C07312=1184.662,313.073,-71.587,-176.592,7.819,148.515
C07313=1184.666,312.825,-71.556,-176.595,7.816,148.515
C07314=1184.670,312.577,-71.525,-176.597,7.813,148.515
C07315=1184.675,312.329,-71.495,-176.599,7.810,148.515
C07316=1184.679,312.081,-71.463,-176.602,7.807,148.515
C07317=1184.683,311.833,-71.432,-176.604,7.804,148.515
C07318=1184.687,311.585,-71.402,-176.607,7.801,148.514
C07319=1184.692,311.337,-71.371,-176.609,7.798,148.515
C07320=1184.696,311.089,-71.340,-176.612,7.795,148.515
C07321=1184.700,310.841,-71.309,-176.615,7.792,148.515
C07322=1184.704,310.593,-71.279,-176.617,7.790,148.514
C07323=1184.709,310.345,-71.248,-176.619,7.787,148.514
C07324=1184.713,310.096,-71.217,-176.622,7.784,148.514
C07325=1184.717,309.849,-71.187,-176.624,7.780,148.514
C07326=1184.721,309.601,-71.156,-176.627,7.777,148.514
C07327=1184.726,309.353,-71.125,-176.630,7.774,148.514
C07328=1184.729,309.104,-71.095,-176.632,7.771,148.514
C07329=1184.734,308.856,-71.064,-176.634,7.769,148.514
C07330=1184.739,308.608,-71.034,-176.637,7.766,148.514
C07331=1184.742,308.360,-71.004,-176.640,7.763,148.514
C07332=1184.746,308.112,-70.973,-176.642,7.760,148.514
C07333=1184.751,307.864,-70.942,-176.645,7.757,148.514
C07334=1184.755,307.616,-70.912,-176.647,7.754,148.514
C07335=1184.760,307.368,-70.881,-176.650,7.751,148.514
C07336=1184.764,307.119,-70.850,-176.652,7.748,148.514
C07337=1184.768,306.871,-70.820,-176.654,7.745,148.514
C07338=1184.772,306.623,-70.790,-176.657,7.742,148.514
C07339=1184.776,306.375,-70.760,-176.660,7.739,148.514
C07340=1184.781,306.128,-70.729,-176.662,7.736,148.514
C07341=1184.785,305.879,-70.698,-176.665,7.733,148.514
C07342=1184.789,305.631,-70.668,-176.667,7.731,148.514
C07343=1184.794,305.383,-70.637,-176.670,7.728,148.514
C07344=1184.798,305.135,-70.607,-176.672,7.725,148.514
C07345=1184.802,304.886,-70.577,-176.675,7.722,148.514
C07346=1184.806,304.638,-70.547,-176.677,7.718,148.514
C07347=1184.810,304.390,-70.516,-176.680,7.715,148.514
C07348=1184.814,304.142,-70.486,-176.682,7.713,148.514
C07349=1184.819,303.894,-70.456,-176.685,7.710,148.514
C07350=1184.823,303.646,-70.426,-176.688,7.707,148.514
C07351=1184.828,303.398,-70.395,-176.690,7.704,148.514
C07352=1184.832,303.150,-70.365,-176.693,7.701,148.514
C07353=1184.836,302.901,-70.334,-176.695,7.698,148.514
C07354=1184.840,302.653,-70.305,-176.697,7.696,148.514
C07355=1184.845,302.405,-70.274,-176.700,7.693,148.514
C07356=1184.849,302.157,-70.244,-176.702,7.689,148.514
C07357=1184.853,301.909,-70.214,-176.705,7.686,148.514
C07358=1184.857,301.661,-70.184,-176.708,7.683,148.514
C07359=1184.861,301.413,-70.154,-176.711,7.680,148.514
C07360=1184.866,301.165,-70.123,-176.713,7.678,148.514
C07361=1184.870,300.916,-70.094,-176.715,7.675,148.514
C07362=1184.874,300.668,-70.063,-176.718,7.672,148.513
C07363=1184.878,300.420,-70.033,-176.720,7.669,148.513
C07364=1184.882,300.172,-70.003,-176.723,7.666,148.513
C07365=1184.887,299.924,-69.973,-176.725,7.664,148.514
C07366=1184.891,299.675,-69.944,-176.728,7.661,148.514
C07367=1184.895,299.428,-69.913,-176.731,7.658,148.514
C07368=1184.900,299.179,-69.883,-176.733,7.655,148.514
C07369=1184.904,298.931,-69.853,-176.736,7.651,148.513
C07370=1184.908,298.683,-69.824,-176.738,7.648,148.513
C07371=1184.913,298.435,-69.794,-176.741,7.646,148.514
C07372=1184.917,298.187,-69.764,-176.743,7.643,148.514
C07373=1184.921,297.939,-69.734,-176.746,7.640,148.514
C07374=1184.926,297.690,-69.704,-176.749,7.637,148.514
C07375=1184.930,297.442,-69.674,-176.751,7.634,148.514
C07376=1184.934,297.194,-69.644,-176.753,7.632,148.513
C07377=1184.938,296.946,-69.615,-176.756,7.629,148.514
C07378=1184.943,296.698,-69.584,-176.759,7.626,148.514
C07379=1184.947,296.450,-69.555,-176.761,7.623,148.514
C07380=1184.951,296.201,-69.525,-176.763,7.621,148.514
C07381=1184.956,295.953,-69.496,-176.766,7.618,148.514
C07382=1184.960,295.705,-69.465,-176.769,7.615,148.514
C07383=1184.964,295.457,-69.436,-176.772,7.612,148.514
C07384=1184.969,295.209,-69.406,-176.774,7.609,148.514
C07385=1184.973,294.960,-69.377,-176.776,7.606,148.514
C07386=1184.977,294.713,-69.347,-176.779,7.603,148.514
C07387=1184.981,294.464,-69.317,-176.781,7.600,148.514
C07388=1184.986,294.216,-69.287,-176.784,7.597,148.514
C07389=1184.990,293.968,-69.258,-176.787,7.594,148.514
C07390=1184.994,293.719,-69.228,-176.789,7.592,148.514
C07391=1184.998,293.471,-69.199,-176.792,7.589,148.514
C07392=1185.002,293.223,-69.169,-176.794,7.586,148.514
C07393=1185.007,292.975,-69.140,-176.797,7.583,148.514
C07394=1185.011,292.727,-69.109,-176.799,7.581,148.514
C07395=1185.015,292.478,-69.080,-176.802,7.578,148.514
C07396=1185.020,292.230,-69.050,-176.805,7.575,148.514
C07397=1185.024,291.982,-69.021,-176.807,7.571,148.514
C07398=1185.028,291.734,-68.991,-176.810,7.568,148.514
C07399=1185.032,291.485,-68.962,-176.812,7.566,148.514
C07400=1185.036,291.237,-68.932,-176.815,7.563,148.514
C07401=1185.040,290.989,-68.903,-176.817,7.560,148.514
C07402=1185.045,290.741,-68.874,-176.820,7.557,148.514
C07403=1185.049,290.493,-68.844,-176.822,7.555,148.514
C07404=1185.054,290.245,-68.815,-176.825,7.552,148.514
C07405=1185.058,289.996,-68.785,-176.828,7.549,148.514
C07406=1185.062,289.748,-68.756,-176.830,7.546,148.514
C07407=1185.066,289.499,-68.727,-176.833,7.544,148.514
C07408=1185.071,289.251,-68.698,-176.835,7.541,148.514
C07409=1185.075,289.003,-68.668,-176.838,7.538,148.514
C07410=1185.080,288.729,-68.635,-176.841,7.535,148.514
C07411=1185.084,288.454,-68.603,-176.843,7.532,148.514
C07412=1185.090,288.179,-68.571,-176.846,7.529,148.514
C07413=1185.094,287.905,-68.539,-176.849,7.525,148.514
C07414=1185.098,287.657,-68.509,-176.852,7.523,148.514
C07415=1185.103,287.408,-68.481,-176.854,7.520,148.514
C07416=1185.107,287.160,-68.451,-176.857,7.517,148.514
C07417=1185.111,286.911,-68.422,-176.860,7.514,148.514
C07418=1185.116,286.663,-68.392,-176.862,7.512,148.515
C07419=1185.120,286.416,-68.363,-176.865,7.509,148.515
C07420=1185.125,286.167,-68.334,-176.867,7.506,148.515
C07421=1185.129,285.918,-68.305,-176.869,7.504,148.515
C07422=1185.133,285.670,-68.275,-176.872,7.501,148.515
C07423=1185.138,285.421,-68.247,-176.875,7.498,148.515
C07424=1185.142,285.174,-68.218,-176.878,7.495,148.515
C07425=1185.146,284.926,-68.189,-176.880,7.493,148.515
C07426=1185.150,284.677,-68.160,-176.883,7.490,148.515
C07427=1185.155,284.429,-68.131,-176.885,7.487,148.515
C07428=1185.159,284.181,-68.102,-176.888,7.484,148.515
C07429=1185.164,283.932,-68.073,-176.890,7.481,148.515
C07430=1185.167,283.684,-68.044,-176.893,7.478,148.515
C07431=1185.171,283.436,-68.014,-176.896,7.475,148.515
C07432=1185.177,283.188,-67.986,-176.898,7.472,148.515
C07433=1185.181,282.940,-67.957,-176.900,7.470,148.515
C07434=1185.185,282.691,-67.928,-176.903,7.467,148.515
C07435=1185.189,282.442,-67.898,-176.906,7.464,148.515
C07436=1185.194,282.195,-67.871,-176.908,7.462,148.515
C07437=1185.198,281.946,-67.841,-176.911,7.459,148.515
C07438=1185.202,281.697,-67.812,-176.914,7.456,148.515
C07439=1185.207,281.450,-67.783,-176.916,7.453,148.515
C07440=1185.211,281.201,-67.755,-176.918,7.451,148.516
C07441=1185.215,280.953,-67.726,-176.921,7.448,148.516
C07442=1185.220,280.705,-67.697,-176.924,7.445,148.516
C07443=1185.224,280.457,-67.669,-176.926,7.443,148.516
C07444=1185.228,280.208,-67.640,-176.929,7.440,148.516
C07445=1185.232,279.960,-67.610,-176.932,7.437,148.516
C07446=1185.237,279.711,-67.582,-176.934,7.435,148.516
C07447=1185.241,279.463,-67.554,-176.937,7.432,148.516
C07448=1185.245,279.215,-67.524,-176.940,7.429,148.516
C07449=1185.250,278.966,-67.496,-176.942,7.426,148.516
C07450=1185.254,278.718,-67.467,-176.944,7.424,148.516
C07451=1185.258,278.470,-67.438,-176.947,7.421,148.516
C07452=1185.263,278.222,-67.411,-176.950,7.418,148.516
C07453=1185.267,277.973,-67.381,-176.952,7.416,148.516
C07454=1185.272,277.725,-67.353,-176.955,7.413,148.516
C07455=1185.276,277.477,-67.325,-176.957,7.410,148.516
C07456=1185.280,277.228,-67.296,-176.960,7.408,148.517
C07457=1185.285,276.980,-67.267,-176.962,7.405,148.517
C07458=1185.289,276.732,-67.239,-176.965,7.402,148.517
C07459=1185.293,276.483,-67.210,-176.968,7.400,148.517
C07460=1185.298,276.235,-67.182,-176.970,7.397,148.517
C07461=1185.302,275.987,-67.153,-176.973,7.394,148.517
C07462=1185.306,275.739,-67.125,-176.975,7.392,148.517
C07463=1185.311,275.490,-67.096,-176.978,7.389,148.517
C07464=1185.314,275.241,-67.068,-176.981,7.386,148.517
C07465=1185.319,274.993,-67.040,-176.983,7.384,148.517
C07466=1185.324,274.745,-67.010,-176.986,7.381,148.517
C07467=1185.328,274.497,-66.983,-176.988,7.378,148.517
C07468=1185.332,274.248,-66.954,-176.991,7.375,148.517
C07469=1185.337,274.000,-66.926,-176.994,7.373,148.518
C07470=1185.341,273.751,-66.897,-176.996,7.370,148.518
C07471=1185.345,273.503,-66.869,-176.999,7.368,148.518
C07472=1185.350,273.255,-66.841,-177.001,7.365,148.518
C07473=1185.354,273.006,-66.813,-177.004,7.362,148.518
C07474=1185.358,272.758,-66.785,-177.006,7.359,148.518
C07475=1185.363,272.509,-66.756,-177.009,7.356,148.518
C07476=1185.367,272.261,-66.728,-177.012,7.353,148.518
C07477=1185.371,272.013,-66.699,-177.014,7.351,148.518
C07478=1185.376,271.765,-66.671,-177.017,7.349,148.518
C07479=1185.380,271.516,-66.642,-177.020,7.346,148.518
C07480=1185.385,271.268,-66.615,-177.022,7.343,148.519
C07481=1185.389,271.019,-66.587,-177.025,7.340,148.519
C07482=1185.394,270.771,-66.559,-177.027,7.337,148.519
C07483=1185.397,270.522,-66.531,-177.029,7.335,148.519
C07484=1185.402,270.274,-66.502,-177.032,7.332,148.519
C07485=1185.406,270.026,-66.474,-177.035,7.330,148.519
C07486=1185.411,269.778,-66.446,-177.038,7.328,148.519
C07487=1185.415,269.529,-66.418,-177.040,7.325,148.519
C07488=1185.419,269.281,-66.390,-177.042,7.322,148.519
C07489=1185.423,269.032,-66.362,-177.045,7.319,148.519
C07490=1185.428,268.784,-66.333,-177.048,7.316,148.519
C07491=1185.433,268.536,-66.306,-177.051,7.315,148.520
C07492=1185.437,268.287,-66.278,-177.053,7.312,148.520
C07493=1185.442,268.039,-66.250,-177.056,7.309,148.520
C07494=1185.445,267.790,-66.222,-177.058,7.306,148.520
C07495=1185.450,267.543,-66.194,-177.061,7.303,148.520
C07496=1185.455,267.293,-66.166,-177.063,7.301,148.520
C07497=1185.459,267.045,-66.138,-177.066,7.299,148.520
C07498=1185.463,266.797,-66.110,-177.069,7.296,148.520
C07499=1185.467,266.549,-66.082,-177.071,7.293,148.520
C07500=1185.472,266.300,-66.054,-177.074,7.290,148.520
C07501=1185.476,266.051,-66.026,-177.077,7.287,148.520
C07502=1185.481,265.803,-65.999,-177.079,7.285,148.520
C07503=1185.485,265.556,-65.971,-177.082,7.283,148.521
C07504=1185.490,265.306,-65.943,-177.084,7.281,148.521
C07505=1185.494,265.058,-65.915,-177.087,7.278,148.521
C07506=1185.498,264.810,-65.887,-177.090,7.275,148.521
C07507=1185.502,264.561,-65.860,-177.092,7.272,148.521
C07508=1185.507,264.313,-65.832,-177.095,7.270,148.521
C07509=1185.512,264.064,-65.804,-177.097,7.268,148.521
C07510=1185.516,263.816,-65.776,-177.100,7.265,148.521
C07511=1185.520,263.568,-65.748,-177.103,7.262,148.521
C07512=1185.524,263.319,-65.721,-177.105,7.259,148.522
C07513=1185.529,263.071,-65.693,-177.108,7.257,148.522
C07514=1185.534,262.798,-65.663,-177.111,7.254,148.522
C07515=1185.539,262.525,-65.632,-177.113,7.251,148.522
C07516=1185.544,262.252,-65.602,-177.117,7.248,148.522
C07517=1185.548,261.979,-65.572,-177.119,7.245,148.522
C07518=1185.552,261.731,-65.545,-177.121,7.243,148.522
C07519=1185.557,261.482,-65.516,-177.125,7.240,148.523
C07520=1185.562,261.233,-65.489,-177.127,7.238,148.523
C07521=1185.566,260.986,-65.461,-177.130,7.235,148.523
C07522=1185.571,260.737,-65.434,-177.132,7.233,148.523
C07523=1185.574,260.489,-65.406,-177.134,7.230,148.523
C07524=1185.579,260.240,-65.379,-177.138,7.227,148.523
C07525=1185.584,259.992,-65.352,-177.140,7.225,148.523
C07526=1185.587,259.743,-65.324,-177.143,7.222,148.523
C07527=1185.592,259.494,-65.297,-177.145,7.220,148.523
C07528=1185.596,259.247,-65.269,-177.148,7.217,148.524
C07529=1185.601,258.998,-65.242,-177.150,7.215,148.524
C07530=1185.605,258.749,-65.214,-177.153,7.212,148.524
C07531=1185.610,258.501,-65.187,-177.156,7.210,148.524
C07532=1185.614,258.253,-65.160,-177.158,7.207,148.524
C07533=1185.619,258.004,-65.132,-177.161,7.204,148.524
C07534=1185.623,257.755,-65.104,-177.163,7.202,148.524
C07535=1185.627,257.507,-65.077,-177.166,7.200,148.525
C07536=1185.632,257.258,-65.050,-177.168,7.198,148.525
C07537=1185.637,257.010,-65.023,-177.171,7.195,148.525
C07538=1185.641,256.762,-64.995,-177.173,7.192,148.525
C07539=1185.645,256.513,-64.968,-177.176,7.190,148.525
C07540=1185.650,256.264,-64.941,-177.179,7.187,148.525
C07541=1185.654,256.016,-64.914,-177.181,7.185,148.525
C07542=1185.658,255.768,-64.887,-177.185,7.182,148.525
C07543=1185.663,255.520,-64.860,-177.187,7.180,148.526
C07544=1185.667,255.271,-64.832,-177.189,7.177,148.526
C07545=1185.671,255.022,-64.805,-177.192,7.175,148.526
C07546=1185.676,254.774,-64.778,-177.195,7.172,148.526
C07547=1185.681,254.525,-64.751,-177.197,7.170,148.526
C07548=1185.685,254.277,-64.724,-177.200,7.167,148.526
C07549=1185.689,254.028,-64.696,-177.202,7.165,148.526
C07550=1185.693,253.780,-64.669,-177.205,7.162,148.526
C07551=1185.698,253.531,-64.642,-177.207,7.160,148.527
C07552=1185.702,253.283,-64.615,-177.210,7.157,148.527
C07553=1185.707,253.034,-64.588,-177.213,7.155,148.527
C07554=1185.712,252.786,-64.561,-177.215,7.152,148.527
C07555=1185.715,252.538,-64.535,-177.218,7.150,148.527
C07556=1185.719,252.289,-64.507,-177.221,7.147,148.527
C07557=1185.724,252.040,-64.480,-177.223,7.145,148.527
C07558=1185.729,251.792,-64.453,-177.226,7.142,148.528
C07559=1185.733,251.543,-64.426,-177.229,7.139,148.528
C07560=1185.737,251.295,-64.399,-177.231,7.137,148.528
C07561=1185.742,251.046,-64.372,-177.234,7.135,148.528
C07562=1185.747,250.798,-64.345,-177.236,7.132,148.528
C07563=1185.751,250.549,-64.318,-177.239,7.130,148.528
C07564=1185.755,250.301,-64.292,-177.242,7.128,148.529
C07565=1185.760,250.053,-64.265,-177.244,7.125,148.529
C07566=1185.765,249.804,-64.238,-177.247,7.123,148.529
C07567=1185.768,249.555,-64.211,-177.250,7.120,148.529
C07568=1185.773,249.306,-64.185,-177.252,7.118,148.529
C07569=1185.778,249.058,-64.157,-177.255,7.115,148.529
C07570=1185.781,248.810,-64.131,-177.257,7.113,148.530
C07571=1185.786,248.561,-64.104,-177.260,7.111,148.530
C07572=1185.791,248.313,-64.077,-177.262,7.108,148.530
C07573=1185.795,248.064,-64.050,-177.265,7.106,148.530
C07574=1185.799,247.816,-64.023,-177.268,7.103,148.530
C07575=1185.804,247.567,-63.997,-177.270,7.101,148.530
C07576=1185.808,247.319,-63.971,-177.273,7.098,148.530
C07577=1185.813,247.070,-63.943,-177.275,7.096,148.531
C07578=1185.818,246.822,-63.916,-177.278,7.093,148.531
C07579=1185.822,246.573,-63.891,-177.281,7.091,148.531
C07580=1185.826,246.324,-63.864,-177.283,7.088,148.531
C07581=1185.830,246.076,-63.837,-177.286,7.086,148.531
C07582=1185.835,245.828,-63.810,-177.289,7.083,148.531
C07583=1185.840,245.578,-63.784,-177.291,7.082,148.532
C07584=1185.844,245.330,-63.757,-177.294,7.079,148.532
C07585=1185.849,245.082,-63.730,-177.296,7.076,148.532
C07586=1185.853,244.833,-63.704,-177.299,7.074,148.532
C07587=1185.857,244.584,-63.677,-177.302,7.072,148.532
C07588=1185.861,244.336,-63.651,-177.305,7.069,148.533
C07589=1185.866,244.087,-63.625,-177.307,7.067,148.533
C07590=1185.870,243.839,-63.598,-177.309,7.065,148.533
C07591=1185.875,243.590,-63.572,-177.312,7.062,148.533
C07592=1185.879,243.342,-63.545,-177.315,7.060,148.533
C07593=1185.884,243.093,-63.518,-177.318,7.057,148.533
C07594=1185.888,242.844,-63.492,-177.320,7.055,148.533
C07595=1185.893,242.596,-63.465,-177.323,7.052,148.534
C07596=1185.897,242.348,-63.440,-177.325,7.050,148.534
C07597=1185.902,242.099,-63.413,-177.328,7.047,148.534
C07598=1185.906,241.850,-63.387,-177.331,7.045,148.534
C07599=1185.911,241.602,-63.360,-177.333,7.043,148.534
C07600=1185.915,241.353,-63.334,-177.336,7.041,148.535
C07601=1185.920,241.105,-63.307,-177.338,7.039,148.535
C07602=1185.924,240.856,-63.282,-177.341,7.036,148.535
C07603=1185.928,240.608,-63.255,-177.344,7.034,148.535
C07604=1185.933,240.359,-63.229,-177.346,7.031,148.535
C07605=1185.937,240.110,-63.202,-177.349,7.029,148.535
C07606=1185.942,239.862,-63.176,-177.352,7.026,148.536
C07607=1185.947,239.613,-63.151,-177.354,7.024,148.536
C07608=1185.951,239.365,-63.124,-177.357,7.022,148.536
C07609=1185.956,239.116,-63.098,-177.360,7.019,148.536
C07610=1185.959,238.868,-63.071,-177.362,7.017,148.536
C07611=1185.964,238.619,-63.046,-177.365,7.015,148.537
C07612=1185.969,238.370,-63.019,-177.367,7.012,148.537
C07613=1185.973,238.122,-62.993,-177.370,7.011,148.537
C07614=1185.977,237.874,-62.967,-177.373,7.008,148.537
C07615=1185.982,237.624,-62.941,-177.375,7.005,148.537
C07616=1185.986,237.376,-62.915,-177.378,7.003,148.538
C07617=1185.991,237.127,-62.889,-177.380,7.001,148.538
C07618=1185.996,236.855,-62.860,-177.383,6.998,148.538
C07619=1186.001,236.585,-62.832,-177.387,6.995,148.538
C07620=1186.006,236.313,-62.804,-177.389,6.993,148.538
C07621=1186.010,236.041,-62.775,-177.392,6.991,148.539
C07622=1186.015,235.792,-62.749,-177.394,6.988,148.539
C07623=1186.019,235.543,-62.723,-177.397,6.986,148.539
C07624=1186.024,235.295,-62.698,-177.400,6.984,148.539
C07625=1186.028,235.047,-62.671,-177.403,6.981,148.539
C07626=1186.033,234.798,-62.645,-177.405,6.979,148.539
C07627=1186.037,234.549,-62.619,-177.408,6.977,148.540
C07628=1186.042,234.301,-62.594,-177.410,6.974,148.540
C07629=1186.046,234.052,-62.568,-177.413,6.972,148.540
C07630=1186.050,233.804,-62.542,-177.415,6.970,148.540
C07631=1186.055,233.554,-62.516,-177.418,6.967,148.541
C07632=1186.060,233.307,-62.490,-177.421,6.965,148.541
C07633=1186.064,233.058,-62.464,-177.424,6.963,148.541
C07634=1186.068,232.809,-62.438,-177.426,6.961,148.541
C07635=1186.073,232.561,-62.412,-177.429,6.959,148.541
C07636=1186.077,232.312,-62.387,-177.432,6.956,148.542
C07637=1186.082,232.063,-62.361,-177.434,6.954,148.542
C07638=1186.087,231.815,-62.335,-177.437,6.952,148.542
C07639=1186.091,231.566,-62.309,-177.439,6.949,148.542
C07640=1186.096,231.318,-62.284,-177.442,6.947,148.543
C07641=1186.100,231.069,-62.258,-177.445,6.944,148.543
C07642=1186.104,230.820,-62.232,-177.447,6.942,148.543
C07643=1186.109,230.572,-62.207,-177.450,6.940,148.543
C07644=1186.113,230.323,-62.181,-177.453,6.938,148.543
C07645=1186.118,230.074,-62.155,-177.455,6.936,148.543
C07646=1186.123,229.826,-62.129,-177.458,6.934,148.544
C07647=1186.127,229.577,-62.104,-177.461,6.931,148.544
C07648=1186.131,229.328,-62.078,-177.463,6.929,148.544
C07649=1186.136,229.080,-62.052,-177.466,6.927,148.544
C07650=1186.141,228.831,-62.027,-177.468,6.924,148.545
C07651=1186.145,228.582,-62.002,-177.471,6.922,148.545
C07652=1186.150,228.334,-61.976,-177.474,6.919,148.545
C07653=1186.154,228.085,-61.951,-177.476,6.918,148.545
C07654=1186.158,227.836,-61.925,-177.479,6.916,148.546
C07655=1186.163,227.588,-61.899,-177.482,6.913,148.546
C07656=1186.167,227.339,-61.874,-177.484,6.911,148.546
C07657=1186.172,227.090,-61.849,-177.487,6.909,148.546
C07658=1186.177,226.842,-61.823,-177.490,6.906,148.546
C07659=1186.181,226.593,-61.798,-177.492,6.904,148.547
C07660=1186.186,226.345,-61.772,-177.495,6.902,148.547
C07661=1186.190,226.095,-61.747,-177.498,6.900,148.547
C07662=1186.194,225.847,-61.721,-177.500,6.897,148.547
C07663=1186.199,225.599,-61.696,-177.503,6.896,148.548
C07664=1186.203,225.350,-61.670,-177.505,6.893,148.548
C07665=1186.208,225.101,-61.646,-177.508,6.891,148.548
C07666=1186.212,224.853,-61.620,-177.511,6.889,148.548
C07667=1186.216,224.604,-61.595,-177.513,6.886,148.548
C07668=1186.221,224.355,-61.570,-177.516,6.884,148.549
C07669=1186.226,224.106,-61.544,-177.518,6.882,148.549
C07670=1186.230,223.858,-61.519,-177.521,6.879,148.549
C07671=1186.235,223.609,-61.494,-177.524,6.878,148.549
C07672=1186.240,223.361,-61.468,-177.526,6.875,148.550
C07673=1186.244,223.112,-61.443,-177.529,6.874,148.550
C07674=1186.248,222.863,-61.418,-177.532,6.871,148.550
C07675=1186.253,222.615,-61.393,-177.534,6.869,148.550
C07676=1186.257,222.365,-61.368,-177.537,6.867,148.551
C07677=1186.262,222.117,-61.342,-177.540,6.864,148.551
C07678=1186.266,221.868,-61.317,-177.542,6.862,148.551
C07679=1186.271,221.620,-61.292,-177.545,6.860,148.551
C07680=1186.275,221.371,-61.267,-177.548,6.857,148.551
C07681=1186.280,221.122,-61.242,-177.550,6.856,148.552
C07682=1186.284,220.873,-61.216,-177.553,6.854,148.552
C07683=1186.289,220.625,-61.192,-177.556,6.851,148.552
C07684=1186.293,220.376,-61.167,-177.558,6.849,148.553
C07685=1186.298,220.128,-61.142,-177.561,6.847,148.553
C07686=1186.302,219.879,-61.116,-177.563,6.845,148.553
C07687=1186.307,219.630,-61.091,-177.567,6.842,148.553
C07688=1186.311,219.381,-61.067,-177.569,6.840,148.553
C07689=1186.316,219.133,-61.042,-177.571,6.838,148.554
C07690=1186.321,218.883,-61.017,-177.575,6.836,148.554
C07691=1186.325,218.635,-60.991,-177.577,6.834,148.554
C07692=1186.329,218.386,-60.967,-177.579,6.832,148.555
C07693=1186.334,218.138,-60.941,-177.582,6.830,148.555
C07694=1186.338,217.889,-60.916,-177.585,6.827,148.555
C07695=1186.343,217.640,-60.892,-177.587,6.825,148.555
C07696=1186.348,217.392,-60.867,-177.590,6.824,148.556
C07697=1186.352,217.143,-60.842,-177.593,6.821,148.556
C07698=1186.357,216.894,-60.818,-177.596,6.819,148.556
C07699=1186.361,216.645,-60.792,-177.598,6.817,148.556
C07700=1186.366,216.397,-60.767,-177.600,6.815,148.556
C07701=1186.370,216.148,-60.743,-177.604,6.812,148.557
C07702=1186.375,215.899,-60.718,-177.606,6.810,148.557
C07703=1186.380,215.651,-60.693,-177.609,6.809,148.557
C07704=1186.384,215.402,-60.668,-177.611,6.806,148.558
C07705=1186.389,215.153,-60.644,-177.614,6.804,148.558
C07706=1186.392,214.904,-60.619,-177.617,6.802,148.558
C07707=1186.397,214.656,-60.594,-177.619,6.800,148.558
C07708=1186.402,214.407,-60.569,-177.622,6.797,148.559
C07709=1186.406,214.158,-60.545,-177.625,6.795,148.559
C07710=1186.411,213.909,-60.520,-177.627,6.793,148.559
C07711=1186.416,213.661,-60.496,-177.630,6.791,148.559
C07712=1186.420,213.412,-60.470,-177.633,6.789,148.560
C07713=1186.424,213.164,-60.446,-177.636,6.787,148.560
C07714=1186.429,212.914,-60.421,-177.638,6.785,148.560
C07715=1186.434,212.665,-60.397,-177.641,6.783,148.561
C07716=1186.438,212.417,-60.373,-177.644,6.780,148.561
C07717=1186.443,212.168,-60.347,-177.646,6.778,148.561
C07718=1186.447,211.919,-60.323,-177.649,6.776,148.561
C07719=1186.452,211.670,-60.299,-177.651,6.775,148.562
C07720=1186.456,211.421,-60.274,-177.654,6.772,148.562
C07721=1186.461,211.173,-60.250,-177.657,6.770,148.562
C07722=1186.466,210.903,-60.223,-177.659,6.768,148.562
C07723=1186.471,210.633,-60.197,-177.663,6.765,148.563
C07724=1186.476,210.362,-60.170,-177.665,6.764,148.563
C07725=1186.481,210.092,-60.143,-177.668,6.761,148.563
C07726=1186.485,209.843,-60.119,-177.671,6.759,148.563
C07727=1186.490,209.594,-60.094,-177.673,6.757,148.564
C07728=1186.494,209.345,-60.070,-177.676,6.754,148.564
C07729=1186.499,209.097,-60.045,-177.679,6.753,148.564
C07730=1186.504,208.848,-60.021,-177.681,6.750,148.565
C07731=1186.508,208.599,-59.996,-177.684,6.749,148.565
C07732=1186.513,208.350,-59.973,-177.687,6.747,148.565
C07733=1186.517,208.101,-59.949,-177.690,6.744,148.566
C07734=1186.522,207.853,-59.924,-177.692,6.742,148.566
C07735=1186.526,207.603,-59.899,-177.695,6.740,148.566
C07736=1186.531,207.355,-59.875,-177.697,6.738,148.566
C07737=1186.536,207.106,-59.851,-177.700,6.737,148.567
C07738=1186.540,206.858,-59.827,-177.703,6.734,148.567
C07739=1186.545,206.608,-59.802,-177.705,6.732,148.567
C07740=1186.549,206.359,-59.778,-177.708,6.730,148.567
C07741=1186.554,206.111,-59.754,-177.711,6.728,148.568
C07742=1186.559,205.862,-59.730,-177.713,6.725,148.568
C07743=1186.563,205.614,-59.705,-177.716,6.724,148.568
C07744=1186.567,205.365,-59.681,-177.719,6.722,148.569
C07745=1186.572,205.115,-59.657,-177.721,6.720,148.569
C07746=1186.577,204.867,-59.633,-177.724,6.718,148.569
C07747=1186.581,204.619,-59.609,-177.727,6.715,148.569
C07748=1186.586,204.370,-59.585,-177.730,6.713,148.570
C07749=1186.590,204.120,-59.561,-177.732,6.712,148.570
C07750=1186.595,203.872,-59.536,-177.735,6.710,148.570
C07751=1186.599,203.623,-59.512,-177.737,6.708,148.571
C07752=1186.604,203.374,-59.489,-177.740,6.706,148.571
C07753=1186.609,203.126,-59.464,-177.743,6.703,148.571
C07754=1186.613,202.876,-59.440,-177.746,6.701,148.572
C07755=1186.617,202.627,-59.417,-177.748,6.699,148.572
C07756=1186.622,202.379,-59.392,-177.750,6.697,148.572
C07757=1186.626,202.131,-59.368,-177.753,6.696,148.572
C07758=1186.632,201.881,-59.344,-177.756,6.693,148.573
C07759=1186.636,201.633,-59.320,-177.759,6.691,148.573
C07760=1186.641,201.384,-59.296,-177.761,6.689,148.573
C07761=1186.645,201.135,-59.273,-177.764,6.687,148.573
C07762=1186.649,200.886,-59.248,-177.766,6.685,148.574
C07763=1186.654,200.637,-59.225,-177.769,6.684,148.574
C07764=1186.659,200.389,-59.200,-177.772,6.681,148.574
C07765=1186.664,200.139,-59.177,-177.775,6.679,148.575
C07766=1186.668,199.891,-59.153,-177.777,6.677,148.575
C07767=1186.673,199.642,-59.130,-177.780,6.675,148.575
C07768=1186.677,199.394,-59.106,-177.783,6.674,148.576
C07769=1186.682,199.145,-59.082,-177.785,6.672,148.576
C07770=1186.686,198.896,-59.058,-177.788,6.669,148.576
C07771=1186.690,198.646,-59.034,-177.791,6.667,148.576
C07772=1186.695,198.398,-59.010,-177.793,6.665,148.577
C07773=1186.700,198.149,-58.986,-177.796,6.663,148.577
C07774=1186.704,197.900,-58.962,-177.799,6.662,148.577
C07775=1186.709,197.651,-58.939,-177.801,6.659,148.578
C07776=1186.714,197.403,-58.915,-177.803,6.658,148.578
C07777=1186.718,197.154,-58.892,-177.807,6.655,148.578
C07778=1186.723,196.905,-58.868,-177.809,6.653,148.579
C07779=1186.727,196.656,-58.844,-177.812,6.651,148.579
C07780=1186.732,196.407,-58.821,-177.815,6.650,148.579
C07781=1186.737,196.158,-58.797,-177.817,6.647,148.579
C07782=1186.741,195.910,-58.773,-177.820,6.646,148.580
C07783=1186.746,195.661,-58.750,-177.822,6.644,148.580
C07784=1186.751,195.412,-58.727,-177.825,6.642,148.580
C07785=1186.755,195.163,-58.703,-177.828,6.639,148.581
C07786=1186.760,194.914,-58.679,-177.831,6.638,148.581
C07787=1186.764,194.665,-58.656,-177.833,6.636,148.581
C07788=1186.769,194.417,-58.632,-177.836,6.634,148.582
C07789=1186.773,194.168,-58.608,-177.838,6.632,148.582
C07790=1186.778,193.919,-58.585,-177.841,6.630,148.582
C07791=1186.783,193.670,-58.562,-177.844,6.628,148.583
C07792=1186.787,193.421,-58.538,-177.846,6.627,148.583
C07793=1186.792,193.172,-58.514,-177.849,6.624,148.583
C07794=1186.797,192.923,-58.491,-177.852,6.622,148.583
C07795=1186.801,192.674,-58.468,-177.854,6.620,148.584
C07796=1186.805,192.426,-58.445,-177.857,6.618,148.584
C07797=1186.810,192.177,-58.421,-177.860,6.616,148.585
C07798=1186.814,191.928,-58.397,-177.862,6.615,148.585
C07799=1186.819,191.679,-58.374,-177.865,6.613,148.585
C07800=1186.824,191.430,-58.351,-177.868,6.611,148.586
C07801=1186.828,191.181,-58.327,-177.870,6.609,148.586
C07802=1186.833,190.932,-58.304,-177.873,6.606,148.586
C07803=1186.838,190.684,-58.281,-177.876,6.604,148.586
C07804=1186.843,190.435,-58.257,-177.878,6.603,148.587
C07805=1186.847,190.187,-58.234,-177.881,6.601,148.587
C07806=1186.852,189.938,-58.211,-177.884,6.599,148.587
C07807=1186.856,189.689,-58.187,-177.886,6.597,148.588
C07808=1186.861,189.439,-58.164,-177.889,6.596,148.588
C07809=1186.866,189.190,-58.141,-177.891,6.593,148.588
C07810=1186.870,188.942,-58.118,-177.894,6.592,148.589
C07811=1186.874,188.693,-58.094,-177.897,6.590,148.589
C07812=1186.879,188.444,-58.071,-177.899,6.588,148.589
C07813=1186.884,188.195,-58.048,-177.902,6.585,148.590
C07814=1186.889,187.946,-58.025,-177.905,6.584,148.590
C07815=1186.893,187.698,-58.002,-177.908,6.582,148.590
C07816=1186.898,187.449,-57.979,-177.910,6.580,148.591
C07817=1186.902,187.199,-57.955,-177.913,6.578,148.591
C07818=1186.907,186.950,-57.932,-177.915,6.576,148.591
C07819=1186.911,186.702,-57.909,-177.918,6.574,148.592
C07820=1186.916,186.453,-57.886,-177.921,6.573,148.592
C07821=1186.921,186.204,-57.864,-177.923,6.571,148.592
C07822=1186.926,185.955,-57.840,-177.926,6.569,148.593
C07823=1186.930,185.706,-57.817,-177.929,6.567,148.593
C07824=1186.935,185.457,-57.794,-177.931,6.565,148.593
C07825=1186.939,185.208,-57.771,-177.934,6.564,148.594
C07826=1186.944,184.938,-57.746,-177.937,6.561,148.594
C07827=1186.949,184.669,-57.721,-177.940,6.559,148.594
C07828=1186.954,184.399,-57.697,-177.943,6.557,148.595
C07829=1186.959,184.130,-57.672,-177.946,6.555,148.595
C07830=1186.964,183.881,-57.649,-177.949,6.553,148.595
C07831=1186.968,183.632,-57.626,-177.951,6.551,148.596
C07832=1186.973,183.383,-57.603,-177.954,6.549,148.596
C07833=1186.978,183.134,-57.579,-177.957,6.548,148.597
C07834=1186.982,182.885,-57.557,-177.959,6.546,148.597
C07835=1186.987,182.637,-57.534,-177.962,6.544,148.597
C07836=1186.991,182.388,-57.511,-177.965,6.542,148.598
C07837=1186.996,182.138,-57.489,-177.967,6.540,148.598
C07838=1187.001,181.889,-57.465,-177.969,6.538,148.598
C07839=1187.006,181.641,-57.443,-177.972,6.536,148.598
C07840=1187.010,181.392,-57.420,-177.975,6.535,148.599
C07841=1187.015,181.143,-57.398,-177.977,6.533,148.599
C07842=1187.019,180.894,-57.374,-177.980,6.531,148.600
C07843=1187.024,180.646,-57.352,-177.983,6.529,148.600
C07844=1187.029,180.396,-57.329,-177.985,6.528,148.600
C07845=1187.033,180.147,-57.306,-177.988,6.526,148.601
C07846=1187.038,179.898,-57.283,-177.991,6.524,148.601
C07847=1187.043,179.650,-57.261,-177.993,6.522,148.601
C07848=1187.047,179.401,-57.238,-177.996,6.520,148.602
C07849=1187.052,179.151,-57.215,-177.999,6.519,148.602
C07850=1187.057,178.903,-57.193,-178.001,6.517,148.602
C07851=1187.062,178.653,-57.170,-178.004,6.515,148.603
C07852=1187.066,178.405,-57.148,-178.007,6.513,148.603
C07853=1187.070,178.156,-57.125,-178.009,6.511,148.603
C07854=1187.075,177.907,-57.103,-178.012,6.510,148.604
C07855=1187.079,177.658,-57.080,-178.015,6.508,148.604
C07856=1187.084,177.409,-57.057,-178.017,6.506,148.604
C07857=1187.089,177.161,-57.035,-178.020,6.504,148.605
C07858=1187.094,176.911,-57.012,-178.022,6.502,148.605
C07859=1187.098,176.662,-56.989,-178.025,6.500,148.605
C07860=1187.103,176.413,-56.967,-178.028,6.499,148.606
C07861=1187.107,176.165,-56.944,-178.030,6.497,148.606
C07862=1187.112,175.915,-56.922,-178.033,6.495,148.606
C07863=1187.117,175.666,-56.900,-178.036,6.493,148.607
C07864=1187.121,175.418,-56.877,-178.038,6.491,148.607
C07865=1187.127,175.169,-56.855,-178.041,6.490,148.608
C07866=1187.131,174.920,-56.832,-178.044,6.488,148.608
C07867=1187.135,174.671,-56.810,-178.046,6.486,148.608
C07868=1187.141,174.422,-56.788,-178.049,6.484,148.609
C07869=1187.145,174.173,-56.765,-178.052,6.483,148.609
C07870=1187.149,173.924,-56.743,-178.054,6.481,148.609
C07871=1187.154,173.675,-56.720,-178.057,6.479,148.610
C07872=1187.158,173.426,-56.698,-178.060,6.477,148.610
C07873=1187.163,173.177,-56.676,-178.062,6.475,148.610
C07874=1187.168,172.928,-56.654,-178.065,6.474,148.611
C07875=1187.172,172.679,-56.631,-178.068,6.472,148.611
C07876=1187.177,172.430,-56.609,-178.070,6.470,148.612
C07877=1187.182,172.181,-56.587,-178.073,6.468,148.612
C07878=1187.187,171.933,-56.564,-178.076,6.467,148.612
C07879=1187.191,171.683,-56.542,-178.078,6.465,148.613
C07880=1187.196,171.434,-56.520,-178.081,6.463,148.613
C07881=1187.201,171.185,-56.498,-178.084,6.461,148.613
C07882=1187.205,170.937,-56.475,-178.087,6.459,148.614
C07883=1187.210,170.688,-56.453,-178.089,6.458,148.614
C07884=1187.215,170.438,-56.431,-178.092,6.456,148.614
C07885=1187.219,170.189,-56.409,-178.095,6.454,148.615
C07886=1187.224,169.940,-56.387,-178.097,6.452,148.615
C07887=1187.228,169.692,-56.365,-178.100,6.450,148.616
C07888=1187.233,169.442,-56.342,-178.103,6.449,148.616
C07889=1187.238,169.194,-56.320,-178.105,6.447,148.616
C07890=1187.242,168.944,-56.298,-178.108,6.445,148.617
C07891=1187.247,168.696,-56.277,-178.111,6.443,148.617
C07892=1187.252,168.446,-56.255,-178.113,6.442,148.617
C07893=1187.257,168.197,-56.232,-178.115,6.441,148.618
C07894=1187.261,167.948,-56.210,-178.118,6.439,148.618
C07895=1187.266,167.700,-56.188,-178.121,6.437,148.619
C07896=1187.270,167.451,-56.166,-178.123,6.435,148.619
C07897=1187.275,167.202,-56.144,-178.127,6.434,148.619
C07898=1187.279,166.953,-56.122,-178.129,6.432,148.620
C07899=1187.284,166.704,-56.100,-178.132,6.430,148.620
C07900=1187.289,166.454,-56.078,-178.135,6.428,148.621
C07901=1187.294,166.206,-56.056,-178.137,6.427,148.621
C07902=1187.298,165.956,-56.034,-178.140,6.425,148.621
C07903=1187.303,165.708,-56.012,-178.143,6.423,148.622
C07904=1187.308,165.459,-55.991,-178.145,6.421,148.622
C07905=1187.312,165.210,-55.969,-178.148,6.420,148.622
C07906=1187.317,164.961,-55.947,-178.151,6.418,148.623
C07907=1187.322,164.712,-55.925,-178.153,6.417,148.623
C07908=1187.326,164.463,-55.903,-178.155,6.415,148.624
C07909=1187.331,164.214,-55.881,-178.158,6.413,148.624
C07910=1187.336,163.965,-55.860,-178.161,6.412,148.624
C07911=1187.340,163.715,-55.838,-178.163,6.410,148.625
C07912=1187.346,163.466,-55.816,-178.166,6.408,148.625
C07913=1187.351,163.218,-55.794,-178.169,6.406,148.625
C07914=1187.355,162.968,-55.772,-178.172,6.404,148.626
C07915=1187.360,162.720,-55.750,-178.174,6.403,148.626
C07916=1187.364,162.470,-55.728,-178.177,6.401,148.627
C07917=1187.369,162.222,-55.707,-178.180,6.399,148.627
C07918=1187.374,161.972,-55.686,-178.182,6.398,148.628
C07919=1187.378,161.723,-55.664,-178.185,6.397,148.628
C07920=1187.383,161.474,-55.642,-178.188,6.395,148.628
C07921=1187.388,161.226,-55.620,-178.190,6.393,148.629
C07922=1187.392,160.976,-55.598,-178.193,6.391,148.629
C07923=1187.397,160.728,-55.578,-178.196,6.390,148.629
C07924=1187.401,160.478,-55.556,-178.198,6.388,148.630
C07925=1187.406,160.230,-55.534,-178.201,6.386,148.630
C07926=1187.411,159.981,-55.512,-178.204,6.384,148.630
C07927=1187.415,159.732,-55.490,-178.206,6.382,148.631
C07928=1187.420,159.482,-55.469,-178.208,6.382,148.631
C07929=1187.425,159.234,-55.448,-178.212,6.380,148.632
C07930=1187.431,158.964,-55.424,-178.214,6.378,148.632
C07931=1187.435,158.696,-55.401,-178.217,6.377,148.633
C07932=1187.441,158.426,-55.378,-178.220,6.374,148.633
C07933=1187.445,158.157,-55.355,-178.223,6.373,148.634
C07934=1187.450,157.909,-55.333,-178.226,6.371,148.634
C07935=1187.455,157.659,-55.312,-178.228,6.370,148.634
C07936=1187.460,157.410,-55.290,-178.231,6.368,148.635
C07937=1187.464,157.162,-55.268,-178.233,6.366,148.635
C07938=1187.468,156.912,-55.248,-178.236,6.364,148.635
C07939=1187.473,156.663,-55.226,-178.239,6.363,148.636
C07940=1187.478,156.414,-55.205,-178.242,6.361,148.636
C07941=1187.483,156.165,-55.183,-178.244,6.359,148.637
C07942=1187.487,155.916,-55.161,-178.247,6.358,148.637
C07943=1187.493,155.667,-55.140,-178.249,6.357,148.638
C07944=1187.497,155.418,-55.119,-178.252,6.355,148.638
C07945=1187.502,155.169,-55.098,-178.255,6.353,148.638
C07946=1187.506,154.920,-55.076,-178.258,6.351,148.639
C07947=1187.511,154.671,-55.055,-178.260,6.350,148.639
C07948=1187.516,154.422,-55.034,-178.263,6.348,148.639
C07949=1187.521,154.173,-55.013,-178.265,6.347,148.640
C07950=1187.525,153.924,-54.991,-178.268,6.345,148.640
C07951=1187.530,153.674,-54.970,-178.271,6.344,148.641
C07952=1187.535,153.426,-54.949,-178.274,6.342,148.641
C07953=1187.539,153.177,-54.928,-178.276,6.340,148.642
C07954=1187.544,152.927,-54.906,-178.279,6.338,148.642
C07955=1187.549,152.678,-54.885,-178.282,6.337,148.642
C07956=1187.554,152.429,-54.864,-178.284,6.336,148.643
C07957=1187.558,152.181,-54.843,-178.286,6.334,148.643
C07958=1187.563,151.931,-54.822,-178.290,6.333,148.644
C07959=1187.568,151.682,-54.800,-178.292,6.331,148.644
C07960=1187.572,151.433,-54.780,-178.295,6.329,148.644
C07961=1187.577,151.184,-54.759,-178.298,6.327,148.645
C07962=1187.582,150.935,-54.737,-178.300,6.326,148.645
C07963=1187.587,150.686,-54.717,-178.302,6.325,148.646
C07964=1187.592,150.437,-54.696,-178.305,6.323,148.646
C07965=1187.596,150.188,-54.674,-178.308,6.321,148.647
C07966=1187.600,149.939,-54.653,-178.311,6.320,148.647
C07967=1187.606,149.689,-54.632,-178.313,6.319,148.647
C07968=1187.610,149.441,-54.611,-178.316,6.317,148.648
C07969=1187.615,149.192,-54.590,-178.318,6.315,148.648
C07970=1187.620,148.943,-54.569,-178.321,6.313,148.648
C07971=1187.624,148.694,-54.548,-178.324,6.312,148.649
C07972=1187.629,148.444,-54.527,-178.327,6.310,148.649
C07973=1187.634,148.195,-54.506,-178.329,6.309,148.650
C07974=1187.638,147.946,-54.486,-178.332,6.307,148.650
C07975=1187.643,147.697,-54.464,-178.334,6.306,148.651
C07976=1187.648,147.448,-54.443,-178.337,6.304,148.651
C07977=1187.653,147.199,-54.423,-178.340,6.302,148.651
C07978=1187.658,146.950,-54.402,-178.342,6.302,148.652
C07979=1187.662,146.700,-54.381,-178.345,6.300,148.652
C07980=1187.667,146.451,-54.360,-178.348,6.298,148.653
C07981=1187.671,146.203,-54.339,-178.350,6.296,148.653
C07982=1187.676,145.953,-54.318,-178.353,6.294,148.654
C07983=1187.681,145.705,-54.297,-178.355,6.293,148.654
C07984=1187.686,145.455,-54.276,-178.358,6.292,148.655
C07985=1187.690,145.206,-54.256,-178.361,6.290,148.655
C07986=1187.696,144.957,-54.235,-178.364,6.289,148.655
C07987=1187.700,144.708,-54.215,-178.366,6.288,148.656
C07988=1187.705,144.459,-54.194,-178.369,6.286,148.656
C07989=1187.709,144.211,-54.173,-178.372,6.284,148.657
C07990=1187.715,143.961,-54.152,-178.375,6.283,148.657
C07991=1187.719,143.712,-54.131,-178.377,6.281,148.657
C07992=1187.724,143.462,-54.110,-178.379,6.280,148.658
C07993=1187.728,143.213,-54.090,-178.382,6.278,148.658
C07994=1187.733,142.964,-54.069,-178.385,6.277,148.659
C07995=1187.738,142.715,-54.048,-178.388,6.275,148.659
C07996=1187.742,142.466,-54.028,-178.390,6.274,148.660
C07997=1187.747,142.217,-54.007,-178.393,6.272,148.660
C07998=1187.752,141.968,-53.987,-178.395,6.271,148.660
C07999=1187.757,141.719,-53.966,-178.399,6.269,148.661
C08000=1187.761,141.470,-53.945,-178.401,6.268,148.661
C08001=1187.766,141.221,-53.925,-178.403,6.266,148.662
C08002=1187.771,140.972,-53.904,-178.406,6.265,148.662
C08003=1187.775,140.723,-53.884,-178.409,6.263,148.663
C08004=1187.781,140.473,-53.863,-178.412,6.261,148.663
C08005=1187.785,140.224,-53.843,-178.414,6.261,148.664
C08006=1187.790,139.975,-53.823,-178.417,6.259,148.664
C08007=1187.795,139.726,-53.802,-178.419,6.257,148.664
C08008=1187.799,139.477,-53.781,-178.422,6.255,148.665
C08009=1187.804,139.228,-53.761,-178.425,6.255,148.665
C08010=1187.809,138.978,-53.740,-178.427,6.253,148.666
C08011=1187.813,138.730,-53.719,-178.430,6.251,148.666
C08012=1187.818,138.480,-53.700,-178.433,6.249,148.666
C08013=1187.823,138.231,-53.679,-178.435,6.249,148.667
C08014=1187.828,137.982,-53.659,-178.438,6.247,148.667
C08015=1187.833,137.733,-53.638,-178.441,6.245,148.668
C08016=1187.837,137.485,-53.618,-178.443,6.244,148.668
C08017=1187.843,137.235,-53.598,-178.446,6.243,148.669
C08018=1187.847,136.986,-53.577,-178.449,6.241,148.669
C08019=1187.851,136.737,-53.557,-178.451,6.239,148.670
C08020=1187.857,136.487,-53.536,-178.454,6.238,148.670
C08021=1187.861,136.238,-53.516,-178.456,6.237,148.670
C08022=1187.866,135.989,-53.496,-178.459,6.235,148.671
C08023=1187.870,135.740,-53.476,-178.462,6.233,148.671
C08024=1187.875,135.491,-53.455,-178.464,6.233,148.672
C08025=1187.880,135.241,-53.435,-178.467,6.231,148.672
C08026=1187.885,134.993,-53.415,-178.470,6.229,148.673
C08027=1187.890,134.744,-53.395,-178.472,6.228,148.673
C08028=1187.894,134.494,-53.375,-178.475,6.227,148.674
C08029=1187.900,134.245,-53.354,-178.478,6.225,148.674
C08030=1187.904,133.996,-53.334,-178.481,6.224,148.675
C08031=1187.909,133.747,-53.314,-178.483,6.223,148.675
C08032=1187.913,133.498,-53.294,-178.486,6.221,148.675
C08033=1187.918,133.249,-53.273,-178.488,6.219,148.676
C08034=1187.923,132.980,-53.252,-178.491,6.218,148.676
C08035=1187.928,132.711,-53.231,-178.494,6.216,148.677
C08036=1187.934,132.443,-53.208,-178.497,6.215,148.677
C08037=1187.938,132.174,-53.187,-178.499,6.214,148.678
C08038=1187.944,131.925,-53.166,-178.502,6.212,148.678
C08039=1187.949,131.676,-53.147,-178.505,6.210,148.679
C08040=1187.953,131.427,-53.126,-178.507,6.209,148.679
C08041=1187.958,131.178,-53.107,-178.510,6.208,148.680
C08042=1187.963,130.929,-53.086,-178.513,6.206,148.680
C08043=1187.967,130.679,-53.067,-178.516,6.205,148.681
C08044=1187.972,130.430,-53.046,-178.518,6.204,148.681
C08045=1187.977,130.181,-53.027,-178.521,6.202,148.681
C08046=1187.982,129.932,-53.007,-178.524,6.200,148.682
C08047=1187.986,129.683,-52.987,-178.526,6.200,148.682
C08048=1187.991,129.433,-52.966,-178.529,6.198,148.683
C08049=1187.997,129.185,-52.947,-178.531,6.196,148.683
C08050=1188.001,128.936,-52.926,-178.534,6.195,148.684
C08051=1188.006,128.686,-52.907,-178.537,6.194,148.684
C08052=1188.011,128.436,-52.887,-178.539,6.192,148.685
C08053=1188.015,128.188,-52.867,-178.542,6.191,148.685
C08054=1188.021,127.939,-52.847,-178.545,6.190,148.686
C08055=1188.025,127.690,-52.827,-178.547,6.188,148.686
C08056=1188.030,127.440,-52.807,-178.550,6.187,148.686
C08057=1188.034,127.191,-52.788,-178.553,6.185,148.687
C08058=1188.040,126.942,-52.768,-178.555,6.184,148.688
C08059=1188.044,126.693,-52.748,-178.558,6.183,148.688
C08060=1188.049,126.443,-52.728,-178.561,6.181,148.689
C08061=1188.053,126.194,-52.708,-178.563,6.180,148.689
C08062=1188.059,125.945,-52.689,-178.566,6.179,148.689
C08063=1188.064,125.696,-52.669,-178.568,6.177,148.690
C08064=1188.068,125.447,-52.649,-178.571,6.176,148.690
C08065=1188.072,125.198,-52.630,-178.574,6.175,148.691
C08066=1188.077,124.949,-52.610,-178.576,6.173,148.691
C08067=1188.082,124.700,-52.590,-178.579,6.171,148.692
C08068=1188.086,124.450,-52.570,-178.582,6.171,148.692
C08069=1188.092,124.201,-52.551,-178.584,6.169,148.693
C08070=1188.097,123.952,-52.531,-178.587,6.167,148.693
C08071=1188.101,123.703,-52.511,-178.590,6.166,148.694
C08072=1188.106,123.454,-52.492,-178.592,6.165,148.694
C08073=1188.111,123.204,-52.472,-178.595,6.163,148.694
C08074=1188.116,122.955,-52.453,-178.598,6.162,148.695
C08075=1188.121,122.706,-52.433,-178.600,6.161,148.695
C08076=1188.125,122.457,-52.413,-178.602,6.160,148.696
C08077=1188.130,122.208,-52.394,-178.606,6.158,148.696
C08078=1188.135,121.959,-52.374,-178.608,6.157,148.697
C08079=1188.140,121.709,-52.355,-178.610,6.156,148.697
C08080=1188.144,121.460,-52.335,-178.614,6.154,148.698
C08081=1188.150,121.211,-52.316,-178.616,6.152,148.698
C08082=1188.154,120.962,-52.297,-178.618,6.152,148.699
C08083=1188.159,120.712,-52.277,-178.622,6.150,148.699
C08084=1188.164,120.464,-52.257,-178.624,6.149,148.700
C08085=1188.168,120.214,-52.238,-178.626,6.147,148.700
C08086=1188.173,119.965,-52.218,-178.630,6.146,148.701
C08087=1188.178,119.716,-52.199,-178.632,6.145,148.701
C08088=1188.182,119.467,-52.179,-178.634,6.143,148.702
C08089=1188.188,119.218,-52.160,-178.638,6.142,148.702
C08090=1188.193,118.968,-52.141,-178.640,6.141,148.703
C08091=1188.197,118.719,-52.121,-178.642,6.139,148.703
C08092=1188.202,118.470,-52.102,-178.645,6.139,148.704
C08093=1188.207,118.220,-52.083,-178.648,6.137,148.704
C08094=1188.212,117.972,-52.063,-178.651,6.135,148.704
C08095=1188.217,117.722,-52.044,-178.653,6.135,148.705
C08096=1188.221,117.473,-52.025,-178.656,6.133,148.705
C08097=1188.226,117.224,-52.005,-178.658,6.132,148.706
C08098=1188.231,116.974,-51.986,-178.661,6.131,148.706
C08099=1188.235,116.726,-51.967,-178.664,6.129,148.707
C08100=1188.240,116.476,-51.947,-178.666,6.128,148.707
C08101=1188.245,116.227,-51.928,-178.669,6.126,148.708
C08102=1188.250,115.978,-51.908,-178.671,6.126,148.708
C08103=1188.255,115.728,-51.890,-178.674,6.124,148.709
C08104=1188.260,115.479,-51.871,-178.677,6.122,148.709
C08105=1188.265,115.229,-51.851,-178.679,6.121,148.710
C08106=1188.269,114.981,-51.832,-178.682,6.120,148.710
C08107=1188.274,114.731,-51.813,-178.685,6.119,148.711
C08108=1188.279,114.482,-51.793,-178.687,6.117,148.711
C08109=1188.283,114.233,-51.774,-178.690,6.116,148.712
C08110=1188.289,113.984,-51.756,-178.693,6.115,148.712
C08111=1188.294,113.734,-51.736,-178.695,6.113,148.713
C08112=1188.298,113.486,-51.717,-178.698,6.113,148.713
C08113=1188.303,113.236,-51.698,-178.701,6.111,148.714
C08114=1188.308,112.987,-51.679,-178.703,6.110,148.714
C08115=1188.313,112.737,-51.660,-178.706,6.109,148.715
C08116=1188.318,112.488,-51.641,-178.709,6.107,148.715
C08117=1188.322,112.239,-51.622,-178.711,6.106,148.716
C08118=1188.327,111.990,-51.602,-178.714,6.105,148.716
C08119=1188.331,111.741,-51.583,-178.716,6.104,148.717
C08120=1188.337,111.491,-51.565,-178.719,6.102,148.717
C08121=1188.341,111.242,-51.546,-178.721,6.101,148.718
C08122=1188.346,110.993,-51.526,-178.725,6.100,148.718
C08123=1188.351,110.743,-51.508,-178.727,6.098,148.719
C08124=1188.356,110.495,-51.489,-178.729,6.097,148.719
C08125=1188.361,110.246,-51.470,-178.733,6.096,148.720
C08126=1188.366,109.996,-51.451,-178.735,6.095,148.720
C08127=1188.371,109.747,-51.432,-178.738,6.094,148.721
C08128=1188.375,109.498,-51.413,-178.740,6.093,148.721
C08129=1188.381,109.248,-51.394,-178.743,6.091,148.722
C08130=1188.385,108.999,-51.375,-178.745,6.090,148.722
C08131=1188.390,108.750,-51.356,-178.748,6.089,148.723
C08132=1188.395,108.501,-51.338,-178.750,6.088,148.723
C08133=1188.400,108.251,-51.318,-178.753,6.086,148.724
C08134=1188.404,108.003,-51.300,-178.756,6.085,148.724
C08135=1188.409,107.753,-51.281,-178.759,6.084,148.725
C08136=1188.414,107.504,-51.262,-178.761,6.082,148.725
C08137=1188.418,107.254,-51.244,-178.764,6.081,148.726
C08138=1188.424,106.986,-51.223,-178.767,6.080,148.726
C08139=1188.430,106.718,-51.203,-178.770,6.079,148.727
C08140=1188.434,106.449,-51.182,-178.772,6.078,148.727
C08141=1188.440,106.181,-51.162,-178.775,6.076,148.728
C08142=1188.445,105.932,-51.144,-178.778,6.075,148.728
C08143=1188.449,105.682,-51.125,-178.781,6.074,148.729
C08144=1188.454,105.433,-51.107,-178.783,6.072,148.729
C08145=1188.460,105.184,-51.087,-178.785,6.071,148.730
C08146=1188.464,104.934,-51.069,-178.789,6.070,148.730
C08147=1188.468,104.686,-51.050,-178.791,6.069,148.731
C08148=1188.474,104.436,-51.032,-178.794,6.068,148.731
C08149=1188.478,104.187,-51.013,-178.796,6.067,148.732
C08150=1188.483,103.938,-50.995,-178.799,6.065,148.732
C08151=1188.488,103.689,-50.976,-178.801,6.064,148.733
C08152=1188.493,103.439,-50.957,-178.804,6.063,148.733
C08153=1188.497,103.190,-50.938,-178.807,6.062,148.734
C08154=1188.503,102.941,-50.920,-178.809,6.060,148.734
C08155=1188.507,102.691,-50.902,-178.812,6.060,148.735
C08156=1188.512,102.442,-50.883,-178.815,6.058,148.735
C08157=1188.517,102.193,-50.864,-178.817,6.058,148.736
C08158=1188.522,101.943,-50.846,-178.820,6.056,148.736
C08159=1188.526,101.695,-50.827,-178.822,6.055,148.737
C08160=1188.532,101.445,-50.809,-178.825,6.054,148.737
C08161=1188.536,101.195,-50.790,-178.828,6.053,148.738
C08162=1188.541,100.947,-50.772,-178.831,6.051,148.739
C08163=1188.547,100.697,-50.753,-178.833,6.050,148.739
C08164=1188.552,100.448,-50.735,-178.836,6.049,148.740
C08165=1188.556,100.199,-50.716,-178.838,6.048,148.740
C08166=1188.560,99.950,-50.698,-178.841,6.046,148.740
C08167=1188.566,99.700,-50.679,-178.844,6.046,148.741
C08168=1188.570,99.450,-50.661,-178.846,6.044,148.741
C08169=1188.575,99.202,-50.642,-178.849,6.043,148.742
C08170=1188.580,98.952,-50.624,-178.852,6.042,148.743
C08171=1188.585,98.703,-50.606,-178.854,6.041,148.743
C08172=1188.590,98.453,-50.588,-178.857,6.039,148.744
C08173=1188.594,98.205,-50.569,-178.860,6.039,148.744
C08174=1188.599,97.955,-50.551,-178.862,6.037,148.745
C08175=1188.604,97.706,-50.533,-178.864,6.036,148.745
C08176=1188.609,97.457,-50.515,-178.868,6.035,148.746
C08177=1188.614,97.207,-50.496,-178.870,6.034,148.746
C08178=1188.619,96.958,-50.478,-178.873,6.032,148.747
C08179=1188.624,96.709,-50.459,-178.875,6.032,148.747
C08180=1188.629,96.460,-50.441,-178.878,6.030,148.748
C08181=1188.633,96.210,-50.423,-178.880,6.029,148.748
C08182=1188.638,95.961,-50.405,-178.884,6.028,148.749
C08183=1188.644,95.711,-50.386,-178.886,6.027,148.749
C08184=1188.648,95.462,-50.368,-178.888,6.026,148.750
C08185=1188.653,95.213,-50.350,-178.891,6.025,148.750
C08186=1188.658,94.963,-50.332,-178.894,6.024,148.751
C08187=1188.662,94.715,-50.313,-178.896,6.022,148.751
C08188=1188.667,94.465,-50.295,-178.898,6.021,148.752
C08189=1188.672,94.216,-50.277,-178.902,6.020,148.753
C08190=1188.677,93.967,-50.259,-178.904,6.019,148.753
C08191=1188.682,93.718,-50.241,-178.907,6.018,148.754
C08192=1188.687,93.468,-50.223,-178.909,6.017,148.754
C08193=1188.692,93.218,-50.205,-178.912,6.016,148.755
C08194=1188.697,92.969,-50.187,-178.914,6.015,148.755
C08195=1188.702,92.720,-50.169,-178.917,6.014,148.756
C08196=1188.707,92.471,-50.151,-178.920,6.012,148.756
C08197=1188.712,92.222,-50.133,-178.922,6.012,148.757
C08198=1188.716,91.973,-50.115,-178.925,6.010,148.757
C08199=1188.721,91.723,-50.096,-178.928,6.009,148.758
C08200=1188.726,91.474,-50.078,-178.930,6.008,148.758
C08201=1188.731,91.224,-50.060,-178.933,6.007,148.759
C08202=1188.736,90.975,-50.042,-178.936,6.005,148.759
C08203=1188.741,90.725,-50.025,-178.938,6.005,148.760
C08204=1188.746,90.476,-50.007,-178.941,6.004,148.760
C08205=1188.751,90.227,-49.989,-178.944,6.003,148.761
C08206=1188.755,89.978,-49.971,-178.946,6.002,148.761
C08207=1188.760,89.729,-49.953,-178.949,6.000,148.762
C08208=1188.765,89.479,-49.935,-178.951,5.999,148.763
C08209=1188.770,89.230,-49.917,-178.954,5.998,148.763
C08210=1188.775,88.980,-49.899,-178.957,5.997,148.764
C08211=1188.780,88.731,-49.882,-178.959,5.997,148.764
C08212=1188.785,88.482,-49.864,-178.962,5.995,148.765
C08213=1188.790,88.232,-49.846,-178.965,5.994,148.765
C08214=1188.794,87.983,-49.828,-178.967,5.993,148.766
C08215=1188.799,87.734,-49.810,-178.970,5.992,148.766
C08216=1188.804,87.485,-49.792,-178.972,5.991,148.767
C08217=1188.809,87.235,-49.775,-178.975,5.990,148.767
C08218=1188.814,86.986,-49.757,-178.977,5.989,148.768
C08219=1188.819,86.737,-49.739,-178.981,5.987,148.769
C08220=1188.824,86.488,-49.721,-178.983,5.987,148.769
C08221=1188.829,86.238,-49.704,-178.986,5.985,148.770
C08222=1188.834,85.989,-49.686,-178.988,5.984,148.770
C08223=1188.839,85.740,-49.668,-178.991,5.984,148.771
C08224=1188.843,85.490,-49.650,-178.993,5.982,148.771
C08225=1188.848,85.241,-49.633,-178.996,5.981,148.772
C08226=1188.852,84.991,-49.615,-178.999,5.980,148.772
C08227=1188.857,84.742,-49.597,-179.001,5.979,148.773
C08228=1188.862,84.492,-49.580,-179.003,5.978,148.773
C08229=1188.867,84.243,-49.562,-179.007,5.977,148.774
C08230=1188.872,83.994,-49.544,-179.009,5.976,148.774
C08231=1188.877,83.744,-49.527,-179.012,5.975,148.775
C08232=1188.882,83.495,-49.509,-179.014,5.974,148.775
C08233=1188.887,83.246,-49.491,-179.017,5.973,148.776
C08234=1188.892,82.997,-49.474,-179.020,5.971,148.776
C08235=1188.897,82.748,-49.456,-179.022,5.971,148.777
C08236=1188.902,82.499,-49.438,-179.024,5.970,148.778
C08237=1188.907,82.249,-49.422,-179.027,5.969,148.778
C08238=1188.912,82.000,-49.404,-179.030,5.968,148.779
C08239=1188.917,81.750,-49.386,-179.033,5.966,148.779
C08240=1188.922,81.501,-49.368,-179.035,5.965,148.780
C08241=1188.926,81.251,-49.352,-179.038,5.965,148.780
C08242=1188.931,80.983,-49.332,-179.041,5.964,148.781
C08243=1188.937,80.714,-49.314,-179.043,5.963,148.781
C08244=1188.942,80.446,-49.294,-179.046,5.961,148.782
C08245=1188.948,80.178,-49.276,-179.049,5.960,148.783
C08246=1188.952,79.929,-49.258,-179.051,5.959,148.783
C08247=1188.957,79.679,-49.241,-179.054,5.958,148.784
C08248=1188.962,79.430,-49.223,-179.057,5.957,148.784
C08249=1188.967,79.180,-49.206,-179.059,5.956,148.785
C08250=1188.971,78.931,-49.188,-179.062,5.956,148.786
C08251=1188.977,78.682,-49.171,-179.065,5.954,148.786
C08252=1188.982,78.432,-49.153,-179.067,5.953,148.787
C08253=1188.986,78.183,-49.137,-179.070,5.953,148.787
C08254=1188.992,77.934,-49.120,-179.073,5.951,148.788
C08255=1188.997,77.685,-49.102,-179.075,5.950,148.788
C08256=1189.001,77.435,-49.085,-179.078,5.949,148.789
C08257=1189.006,77.186,-49.067,-179.080,5.948,148.789
C08258=1189.011,76.936,-49.050,-179.083,5.947,148.790
C08259=1189.016,76.687,-49.033,-179.086,5.946,148.790
C08260=1189.021,76.438,-49.015,-179.088,5.945,148.791
C08261=1189.025,76.188,-48.998,-179.091,5.945,148.792
C08262=1189.030,75.939,-48.980,-179.094,5.943,148.792
C08263=1189.036,75.690,-48.964,-179.096,5.942,148.793
C08264=1189.040,75.440,-48.947,-179.098,5.941,148.793
C08265=1189.045,75.191,-48.929,-179.102,5.940,148.794
C08266=1189.051,74.941,-48.912,-179.104,5.939,148.794
C08267=1189.055,74.692,-48.895,-179.106,5.939,148.795
C08268=1189.060,74.443,-48.877,-179.109,5.937,148.795
C08269=1189.065,74.194,-48.861,-179.112,5.936,148.796
C08270=1189.070,73.944,-48.843,-179.114,5.936,148.797
C08271=1189.075,73.695,-48.827,-179.117,5.934,148.797
C08272=1189.080,73.445,-48.809,-179.120,5.934,148.798
C08273=1189.084,73.196,-48.792,-179.122,5.933,148.798
C08274=1189.089,72.946,-48.775,-179.125,5.931,148.799
C08275=1189.095,72.697,-48.758,-179.127,5.930,148.799
C08276=1189.099,72.448,-48.741,-179.130,5.930,148.800
C08277=1189.105,72.198,-48.723,-179.132,5.928,148.800
C08278=1189.109,71.949,-48.707,-179.135,5.928,148.801
C08279=1189.114,71.699,-48.689,-179.138,5.927,148.802
C08280=1189.119,71.450,-48.673,-179.140,5.925,148.802
C08281=1189.124,71.201,-48.655,-179.143,5.925,148.803
C08282=1189.129,70.952,-48.638,-179.145,5.924,148.803
C08283=1189.134,70.702,-48.621,-179.148,5.923,148.804
C08284=1189.139,70.453,-48.605,-179.151,5.922,148.804
C08285=1189.144,70.203,-48.588,-179.153,5.921,148.805
C08286=1189.149,69.954,-48.571,-179.156,5.921,148.806
C08287=1189.153,69.705,-48.554,-179.159,5.919,148.806
C08288=1189.159,69.456,-48.537,-179.161,5.918,148.807
C08289=1189.163,69.206,-48.520,-179.163,5.917,148.807
C08290=1189.168,68.957,-48.503,-179.167,5.916,148.808
C08291=1189.173,68.707,-48.486,-179.169,5.916,148.808
C08292=1189.179,68.458,-48.469,-179.171,5.915,148.809
C08293=1189.183,68.208,-48.452,-179.175,5.913,148.809
C08294=1189.188,67.959,-48.436,-179.177,5.912,148.810
C08295=1189.193,67.709,-48.419,-179.179,5.912,148.811
C08296=1189.198,67.460,-48.402,-179.181,5.911,148.811
C08297=1189.203,67.211,-48.385,-179.185,5.910,148.812
C08298=1189.208,66.961,-48.368,-179.187,5.909,148.812
C08299=1189.212,66.712,-48.352,-179.189,5.908,148.813
C08300=1189.218,66.463,-48.335,-179.193,5.907,148.813
C08301=1189.222,66.213,-48.318,-179.195,5.906,148.814
C08302=1189.228,65.963,-48.301,-179.197,5.905,148.814
C08303=1189.233,65.715,-48.285,-179.200,5.905,148.815
C08304=1189.237,65.465,-48.268,-179.203,5.903,148.816
C08305=1189.242,65.215,-48.251,-179.205,5.903,148.816
C08306=1189.248,64.966,-48.234,-179.208,5.902,148.817
C08307=1189.252,64.717,-48.218,-179.211,5.900,148.817
C08308=1189.257,64.467,-48.200,-179.213,5.900,148.818
C08309=1189.262,64.218,-48.184,-179.216,5.899,148.818
C08310=1189.267,63.969,-48.167,-179.218,5.898,148.819
C08311=1189.271,63.719,-48.151,-179.221,5.897,148.819
C08312=1189.277,63.470,-48.134,-179.224,5.896,148.820
C08313=1189.282,63.221,-48.117,-179.226,5.896,148.821
C08314=1189.286,62.971,-48.100,-179.228,5.895,148.821
C08315=1189.292,62.722,-48.084,-179.232,5.893,148.822
C08316=1189.297,62.472,-48.068,-179.234,5.893,148.822
C08317=1189.301,62.223,-48.051,-179.236,5.892,148.823
C08318=1189.306,61.974,-48.035,-179.239,5.891,148.824
C08319=1189.311,61.724,-48.017,-179.242,5.890,148.824
C08320=1189.317,61.475,-48.001,-179.244,5.889,148.825
C08321=1189.321,61.226,-47.984,-179.246,5.888,148.825
C08322=1189.326,60.976,-47.968,-179.249,5.888,148.826
C08323=1189.332,60.727,-47.952,-179.252,5.886,148.827
C08324=1189.336,60.477,-47.935,-179.254,5.886,148.827
C08325=1189.341,60.228,-47.918,-179.257,5.885,148.828
C08326=1189.346,59.979,-47.902,-179.260,5.885,148.828
C08327=1189.350,59.729,-47.886,-179.262,5.883,148.829
C08328=1189.356,59.480,-47.869,-179.265,5.882,148.829
C08329=1189.361,59.230,-47.852,-179.267,5.881,148.830
C08330=1189.366,58.981,-47.836,-179.270,5.881,148.831
C08331=1189.371,58.731,-47.820,-179.273,5.880,148.831
C08332=1189.375,58.482,-47.803,-179.275,5.879,148.832
C08333=1189.381,58.233,-47.787,-179.278,5.878,148.832
C08334=1189.386,57.983,-47.771,-179.280,5.877,148.833
C08335=1189.391,57.734,-47.754,-179.283,5.876,148.833
C08336=1189.395,57.484,-47.738,-179.286,5.875,148.834
C08337=1189.401,57.235,-47.722,-179.288,5.874,148.834
C08338=1189.405,56.985,-47.705,-179.291,5.874,148.835
C08339=1189.410,56.737,-47.689,-179.294,5.873,148.836
C08340=1189.416,56.486,-47.673,-179.296,5.872,148.836
C08341=1189.420,56.237,-47.656,-179.299,5.871,148.837
C08342=1189.425,55.988,-47.640,-179.301,5.870,148.837
C08343=1189.430,55.738,-47.624,-179.304,5.869,148.838
C08344=1189.435,55.489,-47.607,-179.307,5.868,148.839
C08345=1189.440,55.240,-47.591,-179.309,5.868,148.839
C08346=1189.445,54.971,-47.574,-179.311,5.867,148.840
C08347=1189.451,54.703,-47.557,-179.315,5.866,148.840
C08348=1189.456,54.434,-47.538,-179.317,5.865,148.841
C08349=1189.462,54.165,-47.521,-179.321,5.864,148.842
C08350=1189.467,53.917,-47.505,-179.323,5.863,148.842
C08351=1189.472,53.666,-47.489,-179.325,5.862,148.843
C08352=1189.477,53.418,-47.472,-179.328,5.862,148.844
C08353=1189.481,53.168,-47.456,-179.330,5.861,148.844
C08354=1189.487,52.919,-47.440,-179.333,5.860,148.845
C08355=1189.491,52.669,-47.424,-179.336,5.859,148.845
C08356=1189.496,52.420,-47.408,-179.338,5.858,148.846
C08357=1189.501,52.170,-47.392,-179.341,5.858,148.846
C08358=1189.506,51.921,-47.376,-179.343,5.857,148.847
C08359=1189.511,51.671,-47.360,-179.346,5.855,148.848
C08360=1189.516,51.422,-47.343,-179.349,5.855,148.848
C08361=1189.521,51.172,-47.327,-179.351,5.854,148.849
C08362=1189.526,50.923,-47.312,-179.354,5.854,148.849
C08363=1189.531,50.673,-47.295,-179.356,5.853,148.850
C08364=1189.536,50.424,-47.280,-179.359,5.851,148.850
C08365=1189.541,50.175,-47.263,-179.362,5.851,148.851
C08366=1189.546,49.925,-47.247,-179.364,5.850,148.852
C08367=1189.551,49.676,-47.231,-179.366,5.849,148.852
C08368=1189.556,49.426,-47.215,-179.369,5.849,148.853
C08369=1189.561,49.177,-47.199,-179.372,5.848,148.854
C08370=1189.565,48.927,-47.183,-179.374,5.847,148.854
C08371=1189.570,48.678,-47.168,-179.377,5.846,148.855
C08372=1189.576,48.429,-47.152,-179.380,5.846,148.855
C08373=1189.580,48.179,-47.135,-179.382,5.845,148.856
C08374=1189.586,47.930,-47.120,-179.384,5.844,148.856
C08375=1189.590,47.680,-47.103,-179.388,5.843,148.857
C08376=1189.596,47.431,-47.088,-179.390,5.842,148.858
C08377=1189.601,47.181,-47.072,-179.392,5.841,148.858
C08378=1189.606,46.931,-47.056,-179.395,5.841,148.859
C08379=1189.611,46.683,-47.040,-179.397,5.840,148.859
C08380=1189.615,46.433,-47.025,-179.400,5.840,148.860
C08381=1189.620,46.183,-47.009,-179.403,5.838,148.860
C08382=1189.625,45.935,-46.993,-179.405,5.837,148.861
C08383=1189.630,45.684,-46.977,-179.408,5.837,148.862
C08384=1189.635,45.435,-46.961,-179.410,5.836,148.862
C08385=1189.641,45.186,-46.945,-179.413,5.835,148.863
C08386=1189.645,44.936,-46.929,-179.415,5.835,148.864
C08387=1189.650,44.687,-46.914,-179.418,5.833,148.864
C08388=1189.655,44.438,-46.898,-179.421,5.833,148.865
C08389=1189.660,44.188,-46.882,-179.423,5.832,148.865
C08390=1189.666,43.938,-46.867,-179.425,5.831,148.866
C08391=1189.671,43.689,-46.850,-179.428,5.831,148.866
C08392=1189.675,43.440,-46.835,-179.431,5.830,148.867
C08393=1189.680,43.190,-46.819,-179.433,5.829,148.868
C08394=1189.685,42.941,-46.804,-179.436,5.828,148.868
C08395=1189.690,42.691,-46.788,-179.439,5.827,148.869
C08396=1189.696,42.441,-46.772,-179.441,5.827,148.870
C08397=1189.700,42.193,-46.757,-179.444,5.826,148.870
C08398=1189.705,41.943,-46.741,-179.446,5.826,148.871
C08399=1189.710,41.693,-46.725,-179.449,5.825,148.871
C08400=1189.716,41.444,-46.709,-179.452,5.823,148.872
C08401=1189.720,41.195,-46.694,-179.454,5.823,148.872
C08402=1189.725,40.945,-46.678,-179.457,5.822,148.873
C08403=1189.730,40.695,-46.663,-179.459,5.821,148.874
C08404=1189.736,40.446,-46.647,-179.462,5.821,148.874
C08405=1189.740,40.196,-46.632,-179.464,5.820,148.875
C08406=1189.745,39.947,-46.616,-179.466,5.820,148.875
C08407=1189.751,39.697,-46.601,-179.470,5.818,148.876
C08408=1189.755,39.448,-46.586,-179.472,5.818,148.877
C08409=1189.760,39.199,-46.569,-179.474,5.817,148.877
C08410=1189.765,38.949,-46.553,-179.477,5.816,148.878
C08411=1189.770,38.700,-46.539,-179.480,5.816,148.879
C08412=1189.775,38.451,-46.523,-179.482,5.815,148.879
C08413=1189.780,38.201,-46.507,-179.485,5.814,148.880
C08414=1189.785,37.952,-46.492,-179.488,5.813,148.880
C08415=1189.790,37.702,-46.476,-179.490,5.812,148.881
C08416=1189.796,37.452,-46.462,-179.493,5.812,148.881
C08417=1189.800,37.203,-46.447,-179.495,5.811,148.882
C08418=1189.805,36.953,-46.431,-179.497,5.810,148.883
C08419=1189.810,36.704,-46.415,-179.500,5.810,148.883
C08420=1189.815,36.454,-46.400,-179.503,5.809,148.884
C08421=1189.820,36.205,-46.384,-179.505,5.809,148.885
C08422=1189.826,35.956,-46.369,-179.507,5.808,148.885
C08423=1189.830,35.706,-46.353,-179.511,5.807,148.886
C08424=1189.835,35.456,-46.338,-179.513,5.806,148.886
C08425=1189.840,35.207,-46.323,-179.515,5.805,148.887
C08426=1189.845,34.958,-46.307,-179.518,5.805,148.888
C08427=1189.851,34.709,-46.292,-179.521,5.804,148.888
C08428=1189.855,34.458,-46.277,-179.523,5.803,148.889
C08429=1189.860,34.209,-46.261,-179.526,5.803,148.889
C08430=1189.865,33.960,-46.246,-179.528,5.802,148.890
C08431=1189.870,33.710,-46.231,-179.531,5.802,148.891
C08432=1189.875,33.461,-46.216,-179.534,5.800,148.891
C08433=1189.881,33.212,-46.200,-179.536,5.800,148.892
C08434=1189.886,32.961,-46.185,-179.539,5.799,148.892
C08435=1189.890,32.712,-46.170,-179.541,5.798,148.893
C08436=1189.896,32.463,-46.154,-179.544,5.798,148.894
C08437=1189.900,32.213,-46.139,-179.546,5.797,148.894
C08438=1189.906,31.964,-46.124,-179.548,5.796,148.895
C08439=1189.911,31.714,-46.110,-179.551,5.796,148.895
C08440=1189.915,31.464,-46.094,-179.554,5.795,148.896
C08441=1189.920,31.215,-46.079,-179.556,5.795,148.897
C08442=1189.925,30.966,-46.063,-179.559,5.794,148.897
C08443=1189.930,30.716,-46.049,-179.562,5.793,148.898
C08444=1189.936,30.467,-46.033,-179.564,5.792,148.899
C08445=1189.940,30.218,-46.018,-179.567,5.791,148.899
C08446=1189.946,29.968,-46.003,-179.569,5.791,148.900
C08447=1189.951,29.718,-45.988,-179.572,5.790,148.900
C08448=1189.955,29.469,-45.973,-179.574,5.789,148.901
C08449=1189.960,29.219,-45.957,-179.577,5.789,148.901
C08450=1189.965,28.950,-45.942,-179.579,5.788,148.902
C08451=1189.971,28.681,-45.925,-179.582,5.788,148.903
C08452=1189.976,28.413,-45.909,-179.585,5.786,148.903
C08453=1189.982,28.144,-45.893,-179.588,5.786,148.904
C08454=1189.987,27.894,-45.878,-179.590,5.785,148.905
C08455=1189.992,27.645,-45.863,-179.593,5.785,148.905
C08456=1189.997,27.396,-45.848,-179.595,5.784,148.906
C08457=1190.003,27.146,-45.833,-179.598,5.784,148.907
C08458=1190.007,26.897,-45.818,-179.600,5.783,148.907
C08459=1190.012,26.647,-45.804,-179.603,5.782,148.908
C08460=1190.018,26.398,-45.788,-179.605,5.782,148.908
C08461=1190.022,26.149,-45.773,-179.608,5.781,148.909
C08462=1190.027,25.899,-45.759,-179.611,5.780,148.910
C08463=1190.033,25.649,-45.743,-179.613,5.779,148.910
C08464=1190.038,25.400,-45.729,-179.616,5.779,148.911
C08465=1190.043,25.150,-45.713,-179.618,5.778,148.911
C08466=1190.048,24.901,-45.699,-179.621,5.777,148.912
C08467=1190.053,24.652,-45.684,-179.624,5.777,148.913
C08468=1190.058,24.402,-45.669,-179.626,5.776,148.913
C08469=1190.063,24.152,-45.654,-179.628,5.775,148.914
C08470=1190.068,23.903,-45.639,-179.631,5.775,148.915
C08471=1190.073,23.653,-45.624,-179.634,5.774,148.915
C08472=1190.078,23.404,-45.609,-179.636,5.773,148.916
C08473=1190.083,23.155,-45.595,-179.638,5.773,148.916
C08474=1190.088,22.905,-45.581,-179.641,5.772,148.917
C08475=1190.093,22.655,-45.565,-179.644,5.772,148.918
C08476=1190.098,22.406,-45.551,-179.646,5.771,148.918
C08477=1190.103,22.157,-45.536,-179.649,5.771,148.919
C08478=1190.108,21.907,-45.521,-179.651,5.770,148.920
C08479=1190.113,21.658,-45.506,-179.654,5.770,148.920
C08480=1190.118,21.408,-45.492,-179.656,5.769,148.921
C08481=1190.123,21.159,-45.477,-179.659,5.768,148.921
C08482=1190.128,20.909,-45.462,-179.661,5.768,148.922
C08483=1190.133,20.659,-45.448,-179.663,5.767,148.923
C08484=1190.138,20.410,-45.433,-179.667,5.766,148.923
C08485=1190.143,20.160,-45.418,-179.669,5.765,148.924
C08486=1190.149,19.910,-45.404,-179.672,5.765,148.925
C08487=1190.153,19.661,-45.389,-179.674,5.764,148.925
C08488=1190.158,19.411,-45.374,-179.677,5.763,148.926
C08489=1190.163,19.162,-45.359,-179.679,5.763,148.926
C08490=1190.168,18.913,-45.345,-179.682,5.762,148.927
C08491=1190.174,18.663,-45.330,-179.684,5.761,148.928
C08492=1190.178,18.413,-45.316,-179.687,5.761,148.928
C08493=1190.183,18.164,-45.301,-179.690,5.760,148.929
C08494=1190.188,17.914,-45.287,-179.692,5.759,148.929
C08495=1190.194,17.665,-45.273,-179.694,5.759,148.930
C08496=1190.199,17.416,-45.257,-179.697,5.758,148.931
C08497=1190.204,17.166,-45.243,-179.700,5.758,148.931
C08498=1190.209,16.916,-45.229,-179.702,5.757,148.932
C08499=1190.214,16.666,-45.214,-179.704,5.757,148.933
C08500=1190.219,16.417,-45.199,-179.707,5.756,148.933
C08501=1190.224,16.168,-45.185,-179.710,5.756,148.934
C08502=1190.228,15.918,-45.171,-179.712,5.755,148.934
C08503=1190.234,15.668,-45.156,-179.715,5.754,148.935
C08504=1190.239,15.419,-45.141,-179.717,5.754,148.936
C08505=1190.244,15.170,-45.127,-179.720,5.753,148.936
C08506=1190.249,14.920,-45.113,-179.722,5.752,148.937
C08507=1190.254,14.670,-45.098,-179.725,5.752,148.938
C08508=1190.259,14.421,-45.084,-179.727,5.751,148.938
C08509=1190.264,14.172,-45.069,-179.730,5.751,148.939
C08510=1190.269,13.922,-45.055,-179.732,5.750,148.939
C08511=1190.274,13.672,-45.041,-179.735,5.750,148.940
C08512=1190.279,13.423,-45.027,-179.737,5.749,148.941
C08513=1190.284,13.173,-45.012,-179.740,5.748,148.941
C08514=1190.290,12.923,-44.997,-179.742,5.748,148.942
C08515=1190.295,12.674,-44.983,-179.745,5.747,148.943
C08516=1190.300,12.425,-44.968,-179.748,5.747,148.943
C08517=1190.305,12.175,-44.954,-179.750,5.746,148.944
C08518=1190.310,11.926,-44.940,-179.752,5.745,148.944
C08519=1190.315,11.676,-44.926,-179.755,5.745,148.945
C08520=1190.320,11.427,-44.911,-179.758,5.744,148.946
C08521=1190.325,11.177,-44.897,-179.760,5.744,148.946
C08522=1190.330,10.927,-44.883,-179.762,5.743,148.947
C08523=1190.335,10.677,-44.869,-179.765,5.743,148.948
C08524=1190.340,10.428,-44.855,-179.768,5.742,148.948
C08525=1190.345,10.179,-44.840,-179.770,5.741,148.949
C08526=1190.350,9.929,-44.826,-179.773,5.741,148.949
C08527=1190.355,9.679,-44.812,-179.775,5.740,148.950
C08528=1190.360,9.430,-44.798,-179.778,5.740,148.951
C08529=1190.366,9.181,-44.784,-179.780,5.739,148.951
C08530=1190.371,8.931,-44.769,-179.783,5.738,148.952
C08531=1190.376,8.681,-44.755,-179.785,5.738,148.953
C08532=1190.381,8.431,-44.741,-179.787,5.738,148.953
C08533=1190.386,8.182,-44.727,-179.790,5.737,148.954
C08534=1190.391,7.933,-44.713,-179.792,5.737,148.954
C08535=1190.396,7.683,-44.698,-179.795,5.736,148.955
C08536=1190.400,7.434,-44.685,-179.798,5.736,148.956
C08537=1190.406,7.185,-44.671,-179.800,5.735,148.956
C08538=1190.411,6.935,-44.657,-179.802,5.735,148.957
C08539=1190.416,6.685,-44.642,-179.805,5.734,148.958
C08540=1190.421,6.435,-44.628,-179.808,5.734,148.958
C08541=1190.426,6.186,-44.614,-179.810,5.733,148.959
C08542=1190.431,5.937,-44.600,-179.812,5.732,148.959
C08543=1190.436,5.687,-44.586,-179.815,5.732,148.960
C08544=1190.441,5.437,-44.571,-179.818,5.731,148.961
C08545=1190.447,5.188,-44.557,-179.820,5.730,148.961
C08546=1190.451,4.938,-44.544,-179.823,5.730,148.962
C08547=1190.456,4.689,-44.530,-179.825,5.729,148.963
C08548=1190.461,4.439,-44.516,-179.828,5.729,148.963
C08549=1190.467,4.190,-44.502,-179.830,5.728,148.964
C08550=1190.472,3.940,-44.488,-179.833,5.728,148.964
C08551=1190.477,3.690,-44.473,-179.835,5.727,148.965
C08552=1190.483,3.441,-44.460,-179.838,5.727,148.966
C08553=1190.487,3.191,-44.446,-179.840,5.726,148.966
C08554=1190.492,2.922,-44.431,-179.843,5.725,148.967
C08555=1190.497,2.653,-44.416,-179.846,5.725,148.968
C08556=1190.503,2.384,-44.401,-179.848,5.724,148.968
C08557=1190.509,2.115,-44.386,-179.851,5.724,148.969
C08558=1190.514,1.865,-44.372,-179.853,5.723,148.970
C08559=1190.519,1.615,-44.358,-179.856,5.723,148.970
C08560=1190.525,1.366,-44.344,-179.859,5.722,148.971
C08561=1190.529,1.117,-44.331,-179.861,5.722,148.972
C08562=1190.534,0.867,-44.316,-179.864,5.721,148.972
C08563=1190.540,0.617,-44.303,-179.866,5.721,148.973
C08564=1190.545,0.368,-44.289,-179.868,5.721,148.974
C08565=1190.550,0.119,-44.275,-179.870,5.720,148.974
C08566=1190.554,-0.131,-44.261,-179.873,5.720,148.975
C08567=1190.560,-0.381,-44.248,-179.876,5.719,148.975
C08568=1190.565,-0.630,-44.234,-179.878,5.719,148.976
C08569=1190.570,-0.880,-44.220,-179.881,5.718,148.977
C08570=1190.575,-1.130,-44.207,-179.883,5.717,148.977
C08571=1190.580,-1.379,-44.193,-179.886,5.717,148.978
C08572=1190.585,-1.629,-44.178,-179.889,5.716,148.979
C08573=1190.591,-1.878,-44.165,-179.891,5.716,148.979
C08574=1190.595,-2.128,-44.152,-179.893,5.715,148.980
C08575=1190.600,-2.377,-44.137,-179.896,5.715,148.981
C08576=1190.606,-2.627,-44.124,-179.899,5.714,148.981
C08577=1190.610,-2.876,-44.110,-179.901,5.714,148.982
C08578=1190.615,-3.127,-44.097,-179.903,5.714,148.982
C08579=1190.621,-3.376,-44.083,-179.906,5.713,148.983
C08580=1190.625,-3.625,-44.069,-179.908,5.713,148.984
C08581=1190.631,-3.875,-44.056,-179.911,5.712,148.984
C08582=1190.636,-4.125,-44.042,-179.913,5.711,148.985
C08583=1190.641,-4.374,-44.029,-179.916,5.711,148.986
C08584=1190.646,-4.624,-44.015,-179.918,5.710,148.986
C08585=1190.651,-4.874,-44.001,-179.921,5.710,148.987
C08586=1190.656,-5.123,-43.988,-179.923,5.709,148.987
C08587=1190.661,-5.373,-43.975,-179.926,5.708,148.988
C08588=1190.667,-5.622,-43.961,-179.928,5.709,148.989
C08589=1190.671,-5.871,-43.947,-179.931,5.708,148.990
C08590=1190.677,-6.121,-43.934,-179.933,5.708,148.990
C08591=1190.682,-6.371,-43.919,-179.935,5.707,148.991
C08592=1190.687,-6.620,-43.907,-179.938,5.707,148.991
C08593=1190.692,-6.870,-43.893,-179.941,5.706,148.992
C08594=1190.697,-7.120,-43.880,-179.943,5.706,148.993
C08595=1190.703,-7.369,-43.866,-179.946,5.705,148.993
C08596=1190.707,-7.619,-43.853,-179.948,5.704,148.994
C08597=1190.713,-7.868,-43.840,-179.950,5.705,148.995
C08598=1190.718,-8.118,-43.825,-179.953,5.704,148.995
C08599=1190.723,-8.367,-43.813,-179.955,5.703,148.996
C08600=1190.728,-8.617,-43.798,-179.958,5.703,148.996
C08601=1190.733,-8.866,-43.786,-179.960,5.702,148.997
C08602=1190.738,-9.116,-43.771,-179.963,5.702,148.998
C08603=1190.743,-9.365,-43.759,-179.966,5.701,148.999
C08604=1190.748,-9.616,-43.745,-179.968,5.701,148.999
C08605=1190.753,-9.864,-43.732,-179.971,5.700,149.000
C08606=1190.758,-10.115,-43.718,-179.973,5.700,149.000
C08607=1190.764,-10.364,-43.705,-179.975,5.700,149.001
C08608=1190.768,-10.614,-43.692,-179.977,5.699,149.002
C08609=1190.774,-10.863,-43.678,-179.980,5.699,149.002
C08610=1190.778,-11.113,-43.665,-179.983,5.698,149.003
C08611=1190.784,-11.362,-43.651,-179.985,5.698,149.004
C08612=1190.789,-11.613,-43.639,-179.988,5.697,149.004
C08613=1190.794,-11.862,-43.625,-179.990,5.696,149.005
C08614=1190.799,-12.112,-43.612,-179.992,5.697,149.005
C08615=1190.805,-12.361,-43.598,-179.995,5.696,149.006
C08616=1190.809,-12.610,-43.585,-179.998,5.696,149.007
C08617=1190.814,-12.860,-43.572,-180.000,5.695,149.007
C08618=1190.820,-13.110,-43.559,179.998,5.694,149.008
C08619=1190.824,-13.360,-43.546,179.995,5.694,149.009
C08620=1190.830,-13.609,-43.532,179.992,5.693,149.009
C08621=1190.834,-13.859,-43.519,179.990,5.693,149.010
C08622=1190.840,-14.108,-43.506,179.988,5.693,149.011
C08623=1190.845,-14.358,-43.492,179.985,5.692,149.011
C08624=1190.850,-14.607,-43.479,179.983,5.692,149.012
C08625=1190.856,-14.857,-43.466,179.980,5.691,149.012
C08626=1190.860,-15.107,-43.453,179.978,5.691,149.013
C08627=1190.866,-15.356,-43.440,179.975,5.690,149.014
C08628=1190.870,-15.606,-43.427,179.972,5.690,149.014
C08629=1190.876,-15.855,-43.413,179.970,5.690,149.015
C08630=1190.881,-16.105,-43.401,179.968,5.689,149.016
C08631=1190.886,-16.355,-43.388,179.966,5.689,149.016
C08632=1190.891,-16.604,-43.375,179.963,5.688,149.017
C08633=1190.896,-16.854,-43.361,179.960,5.688,149.018
C08634=1190.902,-17.103,-43.348,179.958,5.687,149.018
C08635=1190.907,-17.353,-43.335,179.956,5.687,149.019
C08636=1190.911,-17.603,-43.322,179.953,5.687,149.020
C08637=1190.917,-17.852,-43.309,179.951,5.686,149.020
C08638=1190.922,-18.102,-43.296,179.948,5.686,149.021
C08639=1190.927,-18.351,-43.283,179.946,5.685,149.021
C08640=1190.932,-18.600,-43.270,179.943,5.685,149.022
C08641=1190.937,-18.851,-43.257,179.941,5.684,149.023
C08642=1190.942,-19.100,-43.244,179.938,5.685,149.023
C08643=1190.948,-19.349,-43.231,179.936,5.684,149.024
C08644=1190.952,-19.599,-43.218,179.934,5.683,149.025
C08645=1190.957,-19.849,-43.205,179.931,5.683,149.025
C08646=1190.963,-20.098,-43.192,179.928,5.682,149.026
C08647=1190.968,-20.348,-43.179,179.926,5.682,149.027
C08648=1190.973,-20.598,-43.166,179.924,5.682,149.027
C08649=1190.979,-20.847,-43.153,179.921,5.681,149.028
C08650=1190.983,-21.097,-43.140,179.919,5.681,149.029
C08651=1190.988,-21.347,-43.128,179.916,5.680,149.029
C08652=1190.994,-21.596,-43.114,179.914,5.680,149.030
C08653=1190.999,-21.846,-43.102,179.911,5.679,149.030
C08654=1191.004,-22.096,-43.089,179.909,5.679,149.031
C08655=1191.009,-22.345,-43.076,179.907,5.679,149.032
C08656=1191.014,-22.595,-43.063,179.904,5.678,149.032
C08657=1191.019,-22.845,-43.050,179.902,5.678,149.033
C08658=1191.024,-23.114,-43.036,179.899,5.677,149.034
C08659=1191.031,-23.384,-43.023,179.896,5.677,149.034
C08660=1191.036,-23.653,-43.009,179.894,5.676,149.035
C08661=1191.042,-23.924,-42.995,179.891,5.676,149.036
C08662=1191.047,-24.173,-42.982,179.889,5.676,149.036
C08663=1191.052,-24.422,-42.969,179.886,5.676,149.037
C08664=1191.057,-24.671,-42.957,179.884,5.675,149.038
C08665=1191.062,-24.922,-42.943,179.881,5.674,149.038
C08666=1191.067,-25.171,-42.931,179.879,5.674,149.039
C08667=1191.072,-25.420,-42.918,179.876,5.673,149.040
C08668=1191.078,-25.670,-42.905,179.874,5.674,149.040
C08669=1191.082,-25.920,-42.892,179.872,5.673,149.041
C08670=1191.087,-26.169,-42.880,179.869,5.673,149.042
C08671=1191.093,-26.419,-42.867,179.867,5.672,149.042
C08672=1191.099,-26.669,-42.855,179.864,5.672,149.043
C08673=1191.103,-26.919,-42.842,179.862,5.672,149.044
C08674=1191.108,-27.168,-42.829,179.860,5.671,149.044
C08675=1191.113,-27.417,-42.817,179.857,5.671,149.045
C08676=1191.118,-27.667,-42.804,179.854,5.670,149.046
C08677=1191.123,-27.917,-42.791,179.852,5.670,149.046
C08678=1191.129,-28.167,-42.779,179.850,5.670,149.047
C08679=1191.134,-28.416,-42.766,179.847,5.669,149.047
C08680=1191.139,-28.666,-42.753,179.845,5.669,149.048
C08681=1191.144,-28.916,-42.740,179.842,5.668,149.049
C08682=1191.149,-29.165,-42.728,179.839,5.668,149.050
C08683=1191.154,-29.415,-42.716,179.838,5.668,149.050
C08684=1191.160,-29.664,-42.703,179.835,5.667,149.051
C08685=1191.165,-29.913,-42.691,179.833,5.667,149.051
C08686=1191.169,-30.163,-42.678,179.830,5.666,149.052
C08687=1191.175,-30.414,-42.665,179.828,5.666,149.053
C08688=1191.180,-30.663,-42.653,179.826,5.666,149.053
C08689=1191.186,-30.912,-42.640,179.823,5.666,149.054
C08690=1191.191,-31.162,-42.627,179.820,5.665,149.055
C08691=1191.196,-31.412,-42.615,179.818,5.664,149.055
C08692=1191.201,-31.662,-42.603,179.816,5.665,149.056
C08693=1191.206,-31.911,-42.590,179.813,5.664,149.057
C08694=1191.211,-32.161,-42.578,179.811,5.664,149.057
C08695=1191.216,-32.410,-42.566,179.808,5.663,149.058
C08696=1191.221,-32.659,-42.553,179.806,5.662,149.058
C08697=1191.227,-32.909,-42.541,179.804,5.663,149.059
C08698=1191.231,-33.159,-42.528,179.801,5.662,149.060
C08699=1191.237,-33.409,-42.515,179.799,5.662,149.060
C08700=1191.242,-33.659,-42.504,179.796,5.661,149.061
C08701=1191.247,-33.908,-42.491,179.794,5.661,149.062
C08702=1191.252,-34.157,-42.478,179.792,5.661,149.062
C08703=1191.258,-34.407,-42.467,179.789,5.660,149.063
C08704=1191.263,-34.657,-42.454,179.786,5.660,149.064
C08705=1191.267,-34.907,-42.441,179.784,5.659,149.064
C08706=1191.273,-35.157,-42.429,179.782,5.659,149.065
C08707=1191.278,-35.406,-42.416,179.779,5.659,149.066
C08708=1191.283,-35.656,-42.405,179.777,5.659,149.066
C08709=1191.288,-35.905,-42.392,179.775,5.658,149.067
C08710=1191.294,-36.154,-42.379,179.772,5.658,149.067
C08711=1191.299,-36.404,-42.367,179.770,5.658,149.068
C08712=1191.304,-36.654,-42.355,179.767,5.657,149.069
C08713=1191.310,-36.904,-42.343,179.765,5.656,149.069
C08714=1191.314,-37.154,-42.330,179.763,5.657,149.070
C08715=1191.319,-37.404,-42.318,179.760,5.656,149.071
C08716=1191.325,-37.653,-42.306,179.758,5.656,149.071
C08717=1191.330,-37.903,-42.294,179.755,5.655,149.072
C08718=1191.334,-38.152,-42.282,179.753,5.655,149.073
C08719=1191.340,-38.402,-42.270,179.751,5.655,149.073
C08720=1191.345,-38.651,-42.257,179.748,5.654,149.074
C08721=1191.350,-38.901,-42.245,179.745,5.654,149.075
C08722=1191.356,-39.150,-42.233,179.744,5.654,149.075
C08723=1191.361,-39.400,-42.221,179.741,5.654,149.076
C08724=1191.366,-39.650,-42.208,179.738,5.653,149.077
C08725=1191.371,-39.900,-42.196,179.736,5.653,149.077
C08726=1191.377,-40.149,-42.184,179.734,5.653,149.078
C08727=1191.381,-40.398,-42.172,179.731,5.652,149.078
C08728=1191.386,-40.648,-42.160,179.729,5.652,149.079
C08729=1191.392,-40.898,-42.148,179.726,5.651,149.080
C08730=1191.397,-41.148,-42.136,179.724,5.652,149.081
C08731=1191.402,-41.398,-42.123,179.722,5.651,149.081
C08732=1191.407,-41.648,-42.111,179.719,5.650,149.082
C08733=1191.412,-41.897,-42.099,179.717,5.650,149.082
C08734=1191.417,-42.147,-42.087,179.714,5.650,149.083
C08735=1191.422,-42.397,-42.075,179.712,5.649,149.084
C08736=1191.428,-42.646,-42.063,179.710,5.649,149.084
C08737=1191.433,-42.896,-42.051,179.707,5.649,149.085
C08738=1191.438,-43.145,-42.038,179.705,5.649,149.086
C08739=1191.443,-43.395,-42.027,179.703,5.648,149.086
C08740=1191.448,-43.645,-42.015,179.700,5.648,149.087
C08741=1191.453,-43.894,-42.003,179.697,5.647,149.088
C08742=1191.459,-44.144,-41.991,179.695,5.648,149.088
C08743=1191.464,-44.394,-41.979,179.693,5.647,149.089
C08744=1191.469,-44.643,-41.967,179.690,5.646,149.089
C08745=1191.474,-44.893,-41.955,179.688,5.646,149.090
C08746=1191.480,-45.143,-41.943,179.686,5.646,149.091
C08747=1191.485,-45.392,-41.930,179.683,5.646,149.092
C08748=1191.489,-45.642,-41.919,179.681,5.645,149.092
C08749=1191.495,-45.892,-41.907,179.679,5.645,149.093
C08750=1191.501,-46.141,-41.896,179.676,5.645,149.093
C08751=1191.506,-46.390,-41.883,179.673,5.644,149.094
C08752=1191.511,-46.640,-41.872,179.671,5.644,149.095
C08753=1191.516,-46.890,-41.860,179.669,5.644,149.095
C08754=1191.521,-47.140,-41.848,179.667,5.643,149.096
C08755=1191.527,-47.389,-41.835,179.664,5.643,149.097
C08756=1191.531,-47.639,-41.824,179.662,5.643,149.097
C08757=1191.537,-47.889,-41.812,179.660,5.643,149.098
C08758=1191.542,-48.138,-41.800,179.657,5.642,149.099
C08759=1191.547,-48.387,-41.788,179.654,5.642,149.099
C08760=1191.552,-48.637,-41.776,179.652,5.642,149.100
C08761=1191.557,-48.887,-41.765,179.650,5.641,149.100
C08762=1191.563,-49.157,-41.752,179.647,5.641,149.101
C08763=1191.569,-49.427,-41.739,179.645,5.640,149.102
C08764=1191.574,-49.698,-41.727,179.642,5.640,149.103
C08765=1191.580,-49.968,-41.714,179.640,5.640,149.103
C08766=1191.586,-50.218,-41.702,179.637,5.640,149.104
C08767=1191.590,-50.467,-41.690,179.635,5.639,149.105
C08768=1191.595,-50.717,-41.678,179.632,5.639,149.105
C08769=1191.601,-50.967,-41.667,179.630,5.639,149.106
C08770=1191.605,-51.216,-41.655,179.628,5.638,149.107
C08771=1191.611,-51.466,-41.643,179.625,5.638,149.107
C08772=1191.616,-51.716,-41.632,179.623,5.638,149.108
C08773=1191.621,-51.966,-41.620,179.621,5.638,149.108
C08774=1191.627,-52.215,-41.609,179.618,5.637,149.109
C08775=1191.631,-52.464,-41.597,179.616,5.637,149.110
C08776=1191.637,-52.714,-41.585,179.613,5.637,149.111
C08777=1191.642,-52.964,-41.573,179.611,5.636,149.111
C08778=1191.647,-53.214,-41.562,179.608,5.636,149.112
C08779=1191.652,-53.464,-41.550,179.606,5.636,149.112
C08780=1191.657,-53.713,-41.538,179.604,5.636,149.113
C08781=1191.663,-53.963,-41.527,179.602,5.635,149.114
C08782=1191.668,-54.212,-41.516,179.599,5.635,149.114
C08783=1191.673,-54.462,-41.504,179.597,5.635,149.115
C08784=1191.678,-54.712,-41.492,179.594,5.634,149.116
C08785=1191.683,-54.962,-41.481,179.593,5.634,149.116
C08786=1191.689,-55.212,-41.469,179.590,5.634,149.117
C08787=1191.694,-55.461,-41.457,179.587,5.633,149.118
C08788=1191.700,-55.710,-41.446,179.585,5.634,149.118
C08789=1191.704,-55.960,-41.435,179.583,5.633,149.119
C08790=1191.710,-56.210,-41.423,179.580,5.633,149.120
C08791=1191.714,-56.460,-41.411,179.578,5.632,149.120
C08792=1191.720,-56.709,-41.400,179.576,5.633,149.121
C08793=1191.724,-56.959,-41.388,179.573,5.632,149.121
C08794=1191.731,-57.208,-41.377,179.571,5.631,149.122
C08795=1191.735,-57.458,-41.365,179.569,5.632,149.123
C08796=1191.741,-57.708,-41.354,179.566,5.631,149.124
C08797=1191.745,-57.958,-41.342,179.564,5.630,149.124
C08798=1191.751,-58.207,-41.330,179.562,5.631,149.125
C08799=1191.756,-58.456,-41.319,179.559,5.630,149.125
C08800=1191.762,-58.707,-41.308,179.556,5.630,149.126
C08801=1191.766,-58.957,-41.297,179.555,5.630,149.127
C08802=1191.772,-59.207,-41.285,179.552,5.629,149.127
C08803=1191.777,-59.456,-41.274,179.549,5.629,149.128
C08804=1191.782,-59.705,-41.263,179.547,5.629,149.129
C08805=1191.787,-59.955,-41.251,179.545,5.629,149.129
C08806=1191.792,-60.205,-41.240,179.542,5.628,149.130
C08807=1191.797,-60.455,-41.228,179.540,5.628,149.131
C08808=1191.803,-60.704,-41.218,179.538,5.628,149.131
C08809=1191.808,-60.954,-41.206,179.536,5.627,149.132
C08810=1191.813,-61.204,-41.194,179.533,5.628,149.132
C08811=1191.818,-61.453,-41.183,179.531,5.627,149.133
C08812=1191.824,-61.703,-41.172,179.528,5.627,149.134
C08813=1191.829,-61.952,-41.160,179.527,5.627,149.134
C08814=1191.834,-62.203,-41.149,179.524,5.626,149.135
C08815=1191.839,-62.452,-41.138,179.521,5.626,149.136
C08816=1191.844,-62.701,-41.127,179.519,5.626,149.136
C08817=1191.850,-62.951,-41.115,179.517,5.625,149.137
C08818=1191.854,-63.201,-41.104,179.514,5.625,149.138
C08819=1191.860,-63.451,-41.093,179.512,5.625,149.138
C08820=1191.865,-63.700,-41.082,179.510,5.625,149.139
C08821=1191.870,-63.950,-41.070,179.507,5.624,149.140
C08822=1191.876,-64.200,-41.058,179.505,5.624,149.140
C08823=1191.881,-64.449,-41.048,179.503,5.624,149.141
C08824=1191.886,-64.699,-41.037,179.500,5.623,149.141
C08825=1191.891,-64.949,-41.025,179.498,5.624,149.142
C08826=1191.896,-65.199,-41.015,179.496,5.623,149.143
C08827=1191.902,-65.448,-41.004,179.493,5.623,149.144
C08828=1191.907,-65.698,-40.992,179.491,5.623,149.144
C08829=1191.912,-65.948,-40.980,179.489,5.622,149.145
C08830=1191.917,-66.197,-40.970,179.487,5.623,149.145
C08831=1191.923,-66.447,-40.958,179.484,5.622,149.146
C08832=1191.927,-66.697,-40.947,179.482,5.621,149.147
C08833=1191.933,-66.946,-40.937,179.480,5.622,149.147
C08834=1191.938,-67.196,-40.925,179.477,5.621,149.148
C08835=1191.943,-67.446,-40.914,179.474,5.621,149.149
C08836=1191.949,-67.695,-40.903,179.473,5.621,149.149
C08837=1191.954,-67.945,-40.892,179.470,5.621,149.150
C08838=1191.959,-68.195,-40.880,179.467,5.620,149.151
C08839=1191.964,-68.445,-40.870,179.466,5.620,149.151
C08840=1191.969,-68.694,-40.859,179.463,5.620,149.152
C08841=1191.975,-68.945,-40.848,179.460,5.619,149.153
C08842=1191.980,-69.194,-40.837,179.458,5.620,149.153
C08843=1191.985,-69.443,-40.825,179.456,5.619,149.154
C08844=1191.990,-69.694,-40.815,179.454,5.619,149.154
C08845=1191.996,-69.943,-40.803,179.451,5.619,149.155
C08846=1192.001,-70.193,-40.793,179.449,5.618,149.156
C08847=1192.006,-70.442,-40.782,179.447,5.618,149.156
C08848=1192.011,-70.692,-40.771,179.445,5.618,149.157
C08849=1192.017,-70.942,-40.759,179.442,5.617,149.158
C08850=1192.022,-71.191,-40.748,179.440,5.617,149.158
C08851=1192.027,-71.441,-40.738,179.438,5.617,149.159
C08852=1192.032,-71.690,-40.727,179.436,5.617,149.160
C08853=1192.038,-71.941,-40.716,179.433,5.617,149.160
C08854=1192.043,-72.190,-40.704,179.431,5.616,149.161
C08855=1192.048,-72.440,-40.694,179.429,5.617,149.162
C08856=1192.053,-72.690,-40.683,179.426,5.616,149.162
C08857=1192.059,-72.939,-40.673,179.424,5.615,149.163
C08858=1192.064,-73.189,-40.661,179.422,5.616,149.163
C08859=1192.069,-73.439,-40.650,179.419,5.615,149.164
C08860=1192.074,-73.688,-40.639,179.417,5.616,149.165
C08861=1192.079,-73.938,-40.629,179.415,5.615,149.165
C08862=1192.085,-74.187,-40.618,179.412,5.614,149.166
C08863=1192.090,-74.438,-40.607,179.410,5.615,149.167
C08864=1192.096,-74.687,-40.597,179.408,5.614,149.167
C08865=1192.101,-74.937,-40.585,179.405,5.614,149.168
C08866=1192.105,-75.208,-40.574,179.403,5.614,149.169
C08867=1192.112,-75.479,-40.562,179.400,5.614,149.169
C08868=1192.118,-75.750,-40.550,179.398,5.613,149.170
C08869=1192.122,-76.020,-40.538,179.395,5.613,149.171
C08870=1192.129,-76.270,-40.528,179.393,5.613,149.171
C08871=1192.134,-76.520,-40.517,179.391,5.612,149.172
C08872=1192.139,-76.769,-40.506,179.389,5.613,149.173
C08873=1192.144,-77.020,-40.496,179.386,5.612,149.173
C08874=1192.149,-77.269,-40.485,179.383,5.612,149.174
C08875=1192.154,-77.519,-40.474,179.382,5.612,149.175
C08876=1192.160,-77.768,-40.464,179.379,5.611,149.175
C08877=1192.165,-78.018,-40.453,179.377,5.612,149.176
C08878=1192.170,-78.267,-40.442,179.375,5.611,149.176
C08879=1192.176,-78.518,-40.431,179.372,5.611,149.177
C08880=1192.181,-78.767,-40.420,179.370,5.611,149.178
C08881=1192.186,-79.017,-40.410,179.368,5.610,149.178
C08882=1192.192,-79.267,-40.400,179.366,5.610,149.179
C08883=1192.197,-79.516,-40.388,179.363,5.610,149.180
C08884=1192.202,-79.766,-40.378,179.360,5.610,149.180
C08885=1192.207,-80.016,-40.367,179.359,5.610,149.181
C08886=1192.212,-80.265,-40.357,179.356,5.609,149.182
C08887=1192.217,-80.515,-40.346,179.354,5.610,149.182
C08888=1192.223,-80.765,-40.336,179.352,5.609,149.183
C08889=1192.228,-81.015,-40.325,179.349,5.608,149.184
C08890=1192.233,-81.264,-40.314,179.347,5.609,149.184
C08891=1192.238,-81.514,-40.304,179.345,5.608,149.185
C08892=1192.244,-81.764,-40.293,179.343,5.608,149.185
C08893=1192.249,-82.014,-40.283,179.340,5.608,149.186
C08894=1192.254,-82.263,-40.272,179.337,5.608,149.187
C08895=1192.259,-82.513,-40.261,179.336,5.607,149.187
C08896=1192.265,-82.763,-40.251,179.333,5.607,149.188
C08897=1192.270,-83.013,-40.241,179.331,5.607,149.189
C08898=1192.275,-83.262,-40.230,179.329,5.607,149.189
C08899=1192.281,-83.511,-40.219,179.326,5.606,149.190
C08900=1192.286,-83.762,-40.209,179.324,5.607,149.191
C08901=1192.291,-84.011,-40.199,179.322,5.606,149.191
C08902=1192.296,-84.262,-40.188,179.320,5.606,149.192
C08903=1192.302,-84.511,-40.178,179.317,5.606,149.193
C08904=1192.307,-84.761,-40.167,179.315,5.605,149.193
C08905=1192.312,-85.010,-40.156,179.313,5.605,149.194
C08906=1192.317,-85.260,-40.146,179.310,5.605,149.194
C08907=1192.322,-85.510,-40.136,179.308,5.605,149.195
C08908=1192.328,-85.759,-40.126,179.306,5.605,149.196
C08909=1192.333,-86.010,-40.115,179.304,5.605,149.196
C08910=1192.338,-86.258,-40.105,179.301,5.605,149.197
C08911=1192.343,-86.509,-40.094,179.299,5.604,149.198
C08912=1192.349,-86.758,-40.084,179.297,5.604,149.198
C08913=1192.354,-87.008,-40.074,179.294,5.604,149.199
C08914=1192.359,-87.258,-40.063,179.293,5.604,149.199
C08915=1192.365,-87.508,-40.053,179.290,5.603,149.200
C08916=1192.370,-87.758,-40.042,179.288,5.604,149.201
C08917=1192.375,-88.007,-40.033,179.286,5.603,149.201
C08918=1192.380,-88.257,-40.022,179.283,5.602,149.202
C08919=1192.385,-88.507,-40.012,179.281,5.603,149.203
C08920=1192.391,-88.756,-40.002,179.279,5.602,149.203
C08921=1192.396,-89.007,-39.991,179.277,5.602,149.204
C08922=1192.401,-89.256,-39.980,179.274,5.602,149.205
C08923=1192.407,-89.505,-39.970,179.273,5.602,149.205
C08924=1192.411,-89.755,-39.960,179.270,5.602,149.206
C08925=1192.417,-90.005,-39.950,179.267,5.601,149.207
C08926=1192.422,-90.254,-39.939,179.266,5.601,149.207
C08927=1192.427,-90.504,-39.929,179.263,5.601,149.208
C08928=1192.433,-90.754,-39.919,179.261,5.601,149.209
C08929=1192.438,-91.003,-39.908,179.259,5.600,149.209
C08930=1192.443,-91.253,-39.898,179.257,5.601,149.210
C08931=1192.448,-91.503,-39.888,179.254,5.600,149.210
C08932=1192.454,-91.752,-39.878,179.251,5.600,149.211
C08933=1192.459,-92.003,-39.867,179.250,5.600,149.212
C08934=1192.464,-92.252,-39.857,179.247,5.600,149.212
C08935=1192.469,-92.501,-39.848,179.245,5.600,149.213
C08936=1192.475,-92.752,-39.838,179.243,5.599,149.214
C08937=1192.480,-93.002,-39.828,179.241,5.600,149.214
C08938=1192.486,-93.251,-39.817,179.238,5.599,149.215
C08939=1192.491,-93.502,-39.807,179.236,5.599,149.215
C08940=1192.496,-93.751,-39.797,179.234,5.599,149.216
C08941=1192.501,-94.000,-39.787,179.231,5.598,149.217
C08942=1192.506,-94.251,-39.776,179.229,5.598,149.217
C08943=1192.512,-94.500,-39.766,179.227,5.598,149.218
C08944=1192.517,-94.749,-39.757,179.225,5.598,149.219
C08945=1192.522,-95.000,-39.746,179.222,5.597,149.219
C08946=1192.527,-95.249,-39.736,179.220,5.598,149.220
C08947=1192.533,-95.499,-39.726,179.218,5.597,149.220
C08948=1192.538,-95.749,-39.717,179.216,5.597,149.221
C08949=1192.543,-95.999,-39.706,179.213,5.597,149.222
C08950=1192.549,-96.248,-39.696,179.211,5.596,149.222
C08951=1192.554,-96.498,-39.686,179.209,5.597,149.223
C08952=1192.559,-96.747,-39.676,179.206,5.596,149.224
C08953=1192.564,-96.997,-39.666,179.205,5.596,149.224
C08954=1192.570,-97.248,-39.656,179.202,5.596,149.225
C08955=1192.575,-97.497,-39.646,179.200,5.596,149.226
C08956=1192.580,-97.747,-39.636,179.198,5.595,149.226
C08957=1192.585,-97.997,-39.626,179.196,5.596,149.227
C08958=1192.590,-98.246,-39.616,179.193,5.595,149.228
C08959=1192.596,-98.496,-39.607,179.192,5.595,149.228
C08960=1192.602,-98.746,-39.596,179.189,5.595,149.229
C08961=1192.607,-98.996,-39.586,179.186,5.595,149.230
C08962=1192.612,-99.245,-39.576,179.185,5.595,149.230
C08963=1192.618,-99.495,-39.567,179.182,5.594,149.231
C08964=1192.623,-99.745,-39.556,179.180,5.594,149.231
C08965=1192.627,-99.995,-39.546,179.178,5.594,149.232
C08966=1192.633,-100.244,-39.536,179.176,5.594,149.233
C08967=1192.638,-100.494,-39.527,179.173,5.593,149.233
C08968=1192.644,-100.744,-39.517,179.171,5.594,149.234
C08969=1192.649,-100.994,-39.507,179.169,5.593,149.235
C08970=1192.655,-101.264,-39.496,179.167,5.593,149.235
C08971=1192.660,-101.536,-39.486,179.164,5.593,149.236
C08972=1192.666,-101.808,-39.474,179.162,5.593,149.236
C08973=1192.671,-102.080,-39.464,179.160,5.593,149.237
C08974=1192.677,-102.329,-39.454,179.157,5.593,149.238
C08975=1192.682,-102.579,-39.445,179.155,5.592,149.238
C08976=1192.688,-102.829,-39.435,179.153,5.592,149.239
C08977=1192.693,-103.078,-39.425,179.150,5.592,149.240
C08978=1192.698,-103.329,-39.415,179.148,5.592,149.240
C08979=1192.704,-103.578,-39.405,179.146,5.591,149.241
C08980=1192.708,-103.828,-39.395,179.144,5.591,149.241
C08981=1192.714,-104.078,-39.386,179.141,5.591,149.242
C08982=1192.719,-104.327,-39.376,179.139,5.591,149.243
C08983=1192.725,-104.577,-39.366,179.137,5.591,149.243
C08984=1192.729,-104.827,-39.357,179.135,5.591,149.244
C08985=1192.735,-105.077,-39.347,179.132,5.591,149.245
C08986=1192.740,-105.326,-39.337,179.131,5.591,149.245
C08987=1192.746,-105.576,-39.327,179.128,5.590,149.246
C08988=1192.751,-105.825,-39.318,179.126,5.590,149.246
C08989=1192.757,-106.076,-39.308,179.124,5.590,149.247
C08990=1192.762,-106.326,-39.298,179.122,5.590,149.248
C08991=1192.766,-106.575,-39.288,179.119,5.589,149.248
C08992=1192.772,-106.825,-39.279,179.117,5.590,149.249
C08993=1192.777,-107.074,-39.269,179.115,5.589,149.250
C08994=1192.783,-107.325,-39.260,179.113,5.589,149.250
C08995=1192.788,-107.574,-39.250,179.110,5.589,149.251
C08996=1192.794,-107.824,-39.240,179.108,5.588,149.251
C08997=1192.798,-108.074,-39.231,179.106,5.589,149.252
C08998=1192.804,-108.324,-39.221,179.103,5.588,149.253
C08999=1192.809,-108.573,-39.211,179.102,5.588,149.253
C09000=1192.814,-108.823,-39.203,179.099,5.588,149.254
C09001=1192.820,-109.073,-39.192,179.098,5.588,149.255
C09002=1192.825,-109.323,-39.183,179.095,5.588,149.255
C09003=1192.830,-109.572,-39.173,179.093,5.588,149.256
C09004=1192.836,-109.822,-39.164,179.091,5.587,149.257
C09005=1192.841,-110.071,-39.154,179.089,5.588,149.257
C09006=1192.846,-110.321,-39.145,179.086,5.587,149.258
C09007=1192.851,-110.572,-39.135,179.084,5.587,149.258
C09008=1192.856,-110.821,-39.126,179.082,5.587,149.259
C09009=1192.862,-111.071,-39.116,179.080,5.587,149.260
C09010=1192.867,-111.321,-39.107,179.077,5.586,149.260
C09011=1192.872,-111.570,-39.097,179.076,5.586,149.261
C09012=1192.878,-111.820,-39.088,179.073,5.586,149.262
C09013=1192.883,-112.069,-39.078,179.071,5.586,149.262
C09014=1192.889,-112.320,-39.068,179.069,5.586,149.263
C09015=1192.894,-112.569,-39.059,179.067,5.586,149.263
C09016=1192.900,-112.819,-39.049,179.065,5.585,149.264
C09017=1192.905,-113.069,-39.040,179.062,5.586,149.265
C09018=1192.910,-113.318,-39.031,179.060,5.585,149.265
C09019=1192.915,-113.568,-39.021,179.058,5.585,149.266
C09020=1192.921,-113.818,-39.012,179.055,5.585,149.267
C09021=1192.925,-114.067,-39.003,179.054,5.585,149.267
C09022=1192.931,-114.318,-38.993,179.051,5.584,149.268
C09023=1192.936,-114.567,-38.983,179.050,5.584,149.268
C09024=1192.942,-114.818,-38.974,179.047,5.584,149.269
C09025=1192.947,-115.067,-38.965,179.045,5.584,149.270
C09026=1192.952,-115.317,-38.955,179.043,5.584,149.270
C09027=1192.957,-115.567,-38.946,179.041,5.584,149.271
C09028=1192.963,-115.817,-38.937,179.038,5.583,149.271
C09029=1192.967,-116.066,-38.927,179.036,5.584,149.272
C09030=1192.973,-116.316,-38.918,179.034,5.583,149.273
C09031=1192.979,-116.566,-38.909,179.032,5.583,149.273
C09032=1192.983,-116.815,-38.899,179.029,5.583,149.274
C09033=1192.989,-117.065,-38.890,179.028,5.583,149.274
C09034=1192.994,-117.315,-38.881,179.025,5.583,149.275
C09035=1193.000,-117.565,-38.872,179.023,5.583,149.276
C09036=1193.005,-117.815,-38.862,179.021,5.582,149.276
C09037=1193.010,-118.064,-38.853,179.019,5.582,149.277
C09038=1193.016,-118.314,-38.844,179.016,5.582,149.278
C09039=1193.022,-118.564,-38.834,179.014,5.582,149.278
C09040=1193.026,-118.814,-38.825,179.012,5.581,149.279
C09041=1193.032,-119.064,-38.816,179.010,5.582,149.280
C09042=1193.037,-119.313,-38.807,179.008,5.581,149.280
C09043=1193.043,-119.564,-38.798,179.006,5.581,149.281
C09044=1193.047,-119.813,-38.788,179.004,5.581,149.281
C09045=1193.053,-120.063,-38.779,179.002,5.581,149.282
C09046=1193.058,-120.312,-38.770,178.999,5.582,149.283
C09047=1193.064,-120.563,-38.761,178.997,5.581,149.283
C09048=1193.069,-120.812,-38.751,178.995,5.581,149.284
C09049=1193.074,-121.061,-38.743,178.993,5.580,149.284
C09050=1193.079,-121.311,-38.734,178.991,5.581,149.285
C09051=1193.085,-121.561,-38.724,178.989,5.580,149.286
C09052=1193.091,-121.811,-38.715,178.987,5.580,149.286
C09053=1193.095,-122.060,-38.706,178.984,5.580,149.287
C09054=1193.101,-122.310,-38.697,178.982,5.580,149.287
C09055=1193.106,-122.560,-38.687,178.980,5.579,149.288
C09056=1193.112,-122.810,-38.678,178.978,5.580,149.289
C09057=1193.117,-123.060,-38.669,178.975,5.579,149.289
C09058=1193.122,-123.310,-38.661,178.974,5.579,149.290
C09059=1193.127,-123.560,-38.652,178.971,5.579,149.291
C09060=1193.133,-123.809,-38.641,178.970,5.579,149.291
C09061=1193.138,-124.059,-38.633,178.967,5.579,149.292
C09062=1193.143,-124.309,-38.624,178.965,5.579,149.292
C09063=1193.148,-124.559,-38.615,178.963,5.578,149.293
C09064=1193.154,-124.808,-38.606,178.961,5.578,149.293
C09065=1193.159,-125.058,-38.597,178.959,5.579,149.294
C09066=1193.165,-125.308,-38.588,178.957,5.578,149.295
C09067=1193.170,-125.558,-38.579,178.955,5.578,149.295
C09068=1193.175,-125.807,-38.570,178.952,5.577,149.296
C09069=1193.181,-126.057,-38.561,178.950,5.578,149.297
C09070=1193.186,-126.307,-38.552,178.948,5.577,149.297
C09071=1193.191,-126.556,-38.543,178.946,5.577,149.298
C09072=1193.197,-126.807,-38.533,178.943,5.577,149.299
C09073=1193.202,-127.056,-38.525,178.942,5.577,149.299
C09074=1192.781,-127.067,-38.565,178.938,5.580,149.301
C09075=1192.775,-126.818,-38.573,178.939,5.580,149.300
C09076=1192.770,-126.568,-38.582,178.942,5.581,149.300
C09077=1192.764,-126.318,-38.591,178.944,5.581,149.299
C09078=1192.759,-126.068,-38.600,178.946,5.581,149.298
C09079=1192.754,-125.818,-38.609,178.948,5.581,149.298
C09080=1192.749,-125.569,-38.618,178.951,5.581,149.297
C09081=1192.743,-125.318,-38.627,178.952,5.581,149.297
C09082=1192.738,-125.069,-38.636,178.955,5.582,149.296
C09083=1192.733,-124.819,-38.645,178.957,5.582,149.296
C09084=1192.728,-124.569,-38.654,178.959,5.582,149.295
C09085=1192.722,-124.320,-38.662,178.961,5.582,149.294
C09086=1192.717,-124.070,-38.671,178.964,5.582,149.294
C09087=1192.711,-123.820,-38.682,178.966,5.582,149.293
C09088=1192.706,-123.571,-38.690,178.967,5.582,149.292
C09089=1192.701,-123.321,-38.699,178.970,5.582,149.292
C09090=1192.696,-123.071,-38.708,178.971,5.582,149.291
C09091=1192.690,-122.821,-38.717,178.974,5.583,149.291
C09092=1192.684,-122.571,-38.727,178.976,5.583,149.290
C09093=1192.679,-122.321,-38.735,178.978,5.583,149.289
C09094=1192.674,-122.072,-38.745,178.980,5.583,149.289
C09095=1192.669,-121.822,-38.754,178.983,5.584,149.288
C09096=1192.664,-121.572,-38.763,178.984,5.584,149.288
C09097=1192.658,-121.322,-38.772,178.987,5.584,149.287
C09098=1192.653,-121.072,-38.781,178.989,5.584,149.286
C09099=1192.647,-120.823,-38.790,178.991,5.584,149.286
C09100=1192.642,-120.574,-38.799,178.993,5.584,149.285
C09101=1192.637,-120.323,-38.809,178.996,5.585,149.285
C09102=1192.631,-120.074,-38.818,178.998,5.584,149.284
C09103=1192.626,-119.824,-38.827,179.000,5.585,149.283
C09104=1192.621,-119.574,-38.836,179.002,5.585,149.283
C09105=1192.615,-119.324,-38.846,179.004,5.585,149.282
C09106=1192.610,-119.074,-38.855,179.006,5.585,149.281
C09107=1192.605,-118.825,-38.864,179.009,5.585,149.281
C09108=1192.599,-118.574,-38.873,179.010,5.585,149.280
C09109=1192.594,-118.325,-38.883,179.013,5.586,149.279
C09110=1192.589,-118.075,-38.892,179.015,5.586,149.279
C09111=1192.584,-117.826,-38.901,179.017,5.586,149.278
C09112=1192.578,-117.576,-38.911,179.019,5.586,149.278
C09113=1192.573,-117.326,-38.920,179.022,5.587,149.277
C09114=1192.568,-117.076,-38.929,179.023,5.587,149.277
C09115=1192.562,-116.826,-38.938,179.026,5.587,149.276
C09116=1192.557,-116.577,-38.948,179.028,5.587,149.275
C09117=1192.552,-116.327,-38.957,179.030,5.587,149.275
C09118=1192.546,-116.077,-38.966,179.032,5.587,149.274
C09119=1192.541,-115.828,-38.976,179.034,5.587,149.273
C09120=1192.536,-115.578,-38.985,179.037,5.587,149.273
C09121=1192.530,-115.328,-38.994,179.038,5.587,149.272
C09122=1192.525,-115.078,-39.004,179.041,5.588,149.272
C09123=1192.520,-114.829,-39.013,179.043,5.587,149.271
C09124=1192.514,-114.578,-39.022,179.045,5.588,149.270
C09125=1192.509,-114.329,-39.032,179.047,5.588,149.270
C09126=1192.504,-114.079,-39.041,179.049,5.588,149.269
C09127=1192.498,-113.829,-39.050,179.052,5.588,149.268
C09128=1192.494,-113.579,-39.060,179.054,5.588,149.268
C09129=1192.488,-113.329,-39.070,179.056,5.588,149.267
C09130=1192.483,-113.080,-39.079,179.059,5.589,149.267
C09131=1192.478,-112.830,-39.088,179.060,5.589,149.266
C09132=1192.472,-112.580,-39.098,179.063,5.589,149.265
C09133=1192.467,-112.331,-39.107,179.064,5.589,149.265
C09134=1192.462,-112.080,-39.117,179.067,5.590,149.264
C09135=1192.457,-111.831,-39.126,179.069,5.589,149.263
C09136=1192.451,-111.581,-39.136,179.071,5.590,149.263
C09137=1192.446,-111.332,-39.145,179.073,5.590,149.262
C09138=1192.441,-111.082,-39.154,179.076,5.590,149.262
C09139=1192.435,-110.832,-39.164,179.078,5.590,149.261
C09140=1192.430,-110.583,-39.173,179.080,5.590,149.260
C09141=1192.424,-110.332,-39.183,179.083,5.591,149.260
C09142=1192.419,-110.083,-39.192,179.085,5.591,149.259
C09143=1192.414,-109.832,-39.202,179.087,5.592,149.259
C09144=1192.409,-109.583,-39.212,179.089,5.591,149.258
